Destination := value;
TryGetKeyUint := TRUE;
END_METHOD

METHOD TryGetKeyUlint : BOOL
VAR_INPUT
	Key : T_MAXSTRING;
	Destination : REFERENCE TO ULINT;
	Feedback : I_DeserializerFeedback;
END_VAR
VAR
	member : SJsonValue;
	value : ULINT;
	error : I_Error;
END_VAR
IF NOT TryGetMember(Key, member, Feedback) THEN
	RETURN;
END_IF

IF NOT TryReadNumber(member, value) THEN
	error := errorFactory.CreateIncorrectKeyTypeError('ULINT',Key);
	Feedback.LogError(error);
	RETURN;
END_IF

Destination := value;
TryGetKeyUlint := TRUE;
END_METHOD

METHOD TryGetKeyUsint : BOOL
VAR_INPUT
	Key : T_MAXSTRING;
	Destination : REFERENCE TO USINT;
	Feedback : I_DeserializerFeedback;
END_VAR
VAR
	member : SJsonValue;
	value : USINT;
	error : I_Error;
END_VAR
IF NOT TryGetMember(Key, member, Feedback) THEN
	RETURN;
END_IF

IF NOT TryReadNumber(member, value) THEN
	error := errorFactory.CreateIncorrectKeyTypeError('USINT',Key);
	Feedback.LogError(error);
	RETURN;
END_IF

Destination := value;
TryGetKeyUsint := TRUE;
END_METHOD

METHOD TryGetKeyWord : BOOL
VAR_INPUT
	Key : T_MAXSTRING;
	Destination : REFERENCE TO WORD;
	Feedback : I_DeserializerFeedback;
END_VAR
VAR
	member : SJsonValue;
	value : WORD;
	error : I_Error;
END_VAR
IF NOT TryGetMember(Key, member, Feedback) THEN
	RETURN;
END_IF

IF NOT TryReadNumber(member, value) THEN
	error := errorFactory.CreateIncorrectKeyTypeError('USINT',Key);
	Feedback.LogError(error);
	RETURN;
END_IF

Destination := value;
TryGetKeyWord := TRUE;
END_METHOD

METHOD TryGetLint : BOOL
VAR_INPUT
	Destination : REFERENCE TO LINT;
	Feedback : I_DeserializerFeedback;
END_VAR
VAR
	value : LINT;
	error : I_Error;
END_VAR
IF NOT TryReadNumber(root, value) THEN
	error := errorFactory.CreateIncorrectTypeError('LINT');
	Feedback.LogError(error);
	RETURN;
END_IF

Destination := value;
TryGetLint := TRUE;
END_METHOD

METHOD TryGetLreal : BOOL
VAR_INPUT
	Destination : REFERENCE TO LREAL;
	Feedback : I_DeserializerFeedback;
END_VAR
VAR
	value : LREAL;
	error : I_Error;
END_VAR
IF NOT TryReadNumber(root, value) THEN
	error := errorFactory.CreateIncorrectTypeError('LREAL');
	Feedback.LogError(error);
	RETURN;
END_IF

Destination := value;
TryGetLreal := TRUE;
END_METHOD

METHOD TryGetLtime : BOOL
VAR_INPUT
	Destination : REFERENCE TO LTIME;
	Feedback : I_DeserializerFeedback;
END_VAR
VAR
	timeAsString : T_MAXSTRING;
	error : I_Error;
END_VAR
IF NOT jsonParser.IsString(root) THEN
	error := errorFactory.CreateIncorrectTypeError('LTIME');
	Feedback.LogError(error);
	RETURN;
END_IF

timeAsString := jsonParser.GetString(root);
Destination := STRING_TO_LTIME(timeAsString);

TryGetLtime := TRUE;
END_METHOD

METHOD TryGetLword : BOOL
VAR_INPUT
	Destination : REFERENCE TO LWORD;
	Feedback : I_DeserializerFeedback;
END_VAR
VAR
	value : LWORD;
	error : I_Error;
END_VAR
IF NOT TryReadNumber(root, value) THEN
	error := errorFactory.CreateIncorrectTypeError('LWORD');
	Feedback.LogError(error);
	RETURN;
END_IF

Destination := value;
TryGetLword := TRUE;
END_METHOD

METHOD PROTECTED TryGetMember : BOOL
VAR_INPUT
	MemberName : T_MAXSTRING;
	Member : REFERENCE TO SJsonValue;
	Feedback : I_DeserializerFeedback;
END_VAR
VAR
	localMember : SJsonValue;
	error : I_Error;
END_VAR
IF MemberName = '' THEN
	error := errorFactory.CreateInvalidKeyError();
	Feedback.LogError(error);
	RETURN;
END_IF

localMember := jsonParser.FindMember(root, MemberName);

IF localMember = 0 THEN
	error := errorFactory.CreateMissingKeyError(MemberName);
	Feedback.LogError(error);
	RETURN;
END_IF

Member := localMember;
TryGetMember := TRUE;
END_METHOD

METHOD TryGetReal : BOOL
VAR_INPUT
	Destination : REFERENCE TO REAL;
	Feedback : I_DeserializerFeedback;
END_VAR
VAR
	value : REAL;
	error : I_Error;
END_VAR
IF NOT TryReadNumber(root, value) THEN
	error := errorFactory.CreateIncorrectTypeError('REAL');
	Feedback.LogError(error);
	RETURN;
END_IF

Destination := value;
TryGetReal := TRUE;
END_METHOD

METHOD TryGetSint : BOOL
VAR_INPUT
	Destination : REFERENCE TO SINT;
	Feedback : I_DeserializerFeedback;
END_VAR
VAR
	value : SINT;
	error : I_Error;
END_VAR
IF NOT TryReadNumber(root, value) THEN
	error := errorFactory.CreateIncorrectTypeError('SINT');
	Feedback.LogError(error);
	RETURN;
END_IF

Destination := value;
TryGetSint := TRUE;
END_METHOD

METHOD TryGetString : BOOL
VAR_INPUT
	Destination : REFERENCE TO T_MAXSTRING;
	Feedback : I_DeserializerFeedback;
END_VAR
VAR
	error : I_Error;
END_VAR
IF NOT TryReadString(root, Destination) THEN
	error := errorFactory.CreateIncorrectTypeError('STRING');
	Feedback.LogError(error);
	RETURN;
END_IF

TryGetString := TRUE;
END_METHOD

METHOD TryGetStringEx : BOOL
VAR_INPUT
	DestinationAddress : POINTER TO STRING;
	DestinationSize : UDINT;
	Feedback : I_DeserializerFeedback;
END_VAR
VAR
	error : I_Error;
END_VAR
IF NOT TryReadStringEx(root, DestinationAddress, DestinationSize) THEN
	error := errorFactory.CreateIncorrectTypeError('STRING');
	Feedback.LogError(error);
	RETURN;
END_IF

TryGetStringEx := TRUE;
END_METHOD

METHOD TryGetTime : BOOL
VAR_INPUT
	Destination : REFERENCE TO TIME;
	Feedback : I_DeserializerFeedback;
END_VAR
VAR
	timeAsString : T_MAXSTRING;
	error : I_Error;
END_VAR
IF NOT jsonParser.IsString(root) THEN
	error := errorFactory.CreateIncorrectTypeError('TIME');
	Feedback.LogError(error);
	RETURN;
END_IF

timeAsString := jsonParser.GetString(root);
Destination := STRING_TO_TIME(timeAsString);

TryGetTime := TRUE;
END_METHOD

METHOD TryGetTod : BOOL
VAR_INPUT
	Destination : REFERENCE TO TOD;
	Feedback : I_DeserializerFeedback;
END_VAR
VAR
	timeAsString : T_MAXSTRING;
	error : I_Error;
END_VAR
IF NOT jsonParser.IsString(root) THEN
	error := errorFactory.CreateIncorrectTypeError('TOD');
	Feedback.LogError(error);
	RETURN;
END_IF

timeAsString := jsonParser.GetString(root);
Destination := STRING_TO_TOD(timeAsString);

TryGetTod := TRUE;
END_METHOD

METHOD TryGetUdint : BOOL
VAR_INPUT
	Destination : REFERENCE TO UDINT;
	Feedback : I_DeserializerFeedback;
END_VAR
VAR
	value : UDINT;
	error : I_Error;
END_VAR
IF NOT TryReadNumber(root, value) THEN
	error := errorFactory.CreateIncorrectTypeError('UDINT');
	Feedback.LogError(error);
	RETURN;
END_IF

Destination := value;
TryGetUdint := TRUE;
END_METHOD

METHOD TryGetUint : BOOL
VAR_INPUT
	Destination : REFERENCE TO UINT;
	Feedback : I_DeserializerFeedback;
END_VAR
VAR
	value : UINT;
	error : I_Error;
END_VAR
IF NOT TryReadNumber(root, value) THEN
	error := errorFactory.CreateIncorrectTypeError('UINT');
	Feedback.LogError(error);
	RETURN;
END_IF

Destination := value;
TryGetUint := TRUE;
END_METHOD

METHOD TryGetUlint : BOOL
VAR_INPUT
	Destination : REFERENCE TO ULINT;
	Feedback : I_DeserializerFeedback;
END_VAR
VAR
	value : ULINT;
	error : I_Error;
END_VAR
IF NOT TryReadNumber(root, value) THEN
	error := errorFactory.CreateIncorrectTypeError('ULINT');
	Feedback.LogError(error);
	RETURN;
END_IF

Destination := value;
TryGetUlint := TRUE;
END_METHOD

METHOD TryGetUsint : BOOL
VAR_INPUT
	Destination : REFERENCE TO USINT;
	Feedback : I_DeserializerFeedback;
END_VAR
VAR
	value : USINT;
	error : I_Error;
END_VAR
IF NOT TryReadNumber(root, value) THEN
	error := errorFactory.CreateIncorrectTypeError('USINT');
	Feedback.LogError(error);
	RETURN;
END_IF

Destination := value;
TryGetUsint := TRUE;
END_METHOD

METHOD TryGetWord : BOOL
VAR_INPUT
	Destination : REFERENCE TO WORD;
	Feedback : I_DeserializerFeedback;
END_VAR
VAR
	value : WORD;
	error : I_Error;
END_VAR
IF NOT TryReadNumber(root, value) THEN
	error := errorFactory.CreateIncorrectTypeError('WORD');
	Feedback.LogError(error);
	RETURN;
END_IF

Destination := value;
TryGetWord := TRUE;
END_METHOD

METHOD PROTECTED TryReadBool : BOOL
VAR_INPUT
	JsonValue : SJsonValue;
	Destination : ANY;
END_VAR
VAR
	_BOOL : BOOL;
END_VAR
IF jsonValue = 0 THEN
	RETURN;
END_IF

IF jsonParser.IsBool(jsonValue) THEN
	_BOOL := jsonParser.GetBool(jsonValue);
	TryReadBool := TryConvert_BOOL_TO_DESTINATION(_BOOL,Destination);
	RETURN;
END_IF
END_METHOD

METHOD PROTECTED TryReadNumber : BOOL
VAR_INPUT
	JsonValue : SJsonValue;
	Destination : ANY;
END_VAR
VAR
	_DINT : DINT;
	_LINT : LINT;
	_UDINT : UDINT;
	_ULINT : ULINT;
	_LREAL : LREAL;
END_VAR
IF jsonValue = 0 THEN
	RETURN;
END_IF

IF jsonParser.IsInt(jsonValue) THEN
	_DINT := jsonParser.GetInt(jsonValue);
	TryReadNumber := TryConvert_DINT_TO_DESTINATION(_DINT,Destination);
	RETURN;
END_IF

IF jsonParser.IsInt64(jsonValue) THEN
	_LINT := jsonParser.GetInt64(jsonValue);
	TryReadNumber := TryConvert_LINT_TO_DESTINATION(_LINT,Destination);
	RETURN;
END_IF

IF jsonParser.IsUInt(jsonValue) THEN
	_UDINT := jsonParser.GetUInt(jsonValue);
	TryReadNumber := TryConvert_UDINT_TO_DESTINATION(_UDINT,Destination);
	RETURN;
END_IF

IF jsonParser.IsUInt64(jsonValue) THEN
	_ULINT := jsonParser.GetUInt64(jsonValue);
	TryReadNumber := TryConvert_ULINT_TO_DESTINATION(_ULINT,Destination);
	RETURN;
END_IF

IF jsonParser.IsDouble(jsonValue) THEN
	_LREAL := jsonParser.GetDouble(jsonValue);
	TryReadNumber := TryConvert_LREAL_TO_DESTINATION(_LREAL,Destination);
	RETURN;
END_IF
END_METHOD

METHOD PROTECTED TryReadString : BOOL
VAR_INPUT
	JsonValue : SJsonValue;
	Destination : REFERENCE TO T_MAXSTRING;
END_VAR
IF jsonValue = 0 THEN
	RETURN;
END_IF

IF jsonParser.IsString(jsonValue) THEN
	IF (jsonParser.CopyString(jsonValue,Destination,DINT_TO_UDINT(SIZEOF(Destination))) > 0) THEN;
		TryReadString := TRUE;
		RETURN;
	END_IF
END_IF
END_METHOD

METHOD PROTECTED TryReadStringEx : BOOL
VAR_INPUT
	JsonValue : SJsonValue;
	DestinationAddress : POINTER TO STRING;
	DestinationSize : UDINT;
END_VAR
IF jsonValue = 0 THEN
	RETURN;
END_IF

IF jsonParser.IsString(jsonValue) THEN
	IF (jsonParser.CopyString(jsonValue,DestinationAddress^,DestinationSize) > 0) THEN;
		TryReadStringEx := TRUE;
		RETURN;
	END_IF
END_IF
END_METHOD

END_FUNCTION_BLOCK

// ---- mobject-json/_Internal/JsonDeserializerForwardEnumerator/JsonDeserializerArrayForwardEnumerator.TcPOU
{attribute 'linkalways'} 
{attribute 'no_explicit_call' := 'This FB is a CLASS and must be accessed using methods or properties'}
{attribute 'enable_dynamic_creation'}
FUNCTION_BLOCK JsonDeserializerArrayForwardEnumerator EXTENDS Disposable IMPLEMENTS I_DeserializerArrayForwardEnumerator, I_EventHandler
VAR
	parent : I_JsonDeserializer;
	jsonParser : REFERENCE TO JsonDomParser;
	root : SJsonValue;
	garbageCollector : I_DeserializerGarbageCollector;
	nullNode : I_Deserializer;
	moveNextCalled : BOOL := FALSE;
	invalid : BOOL := FALSE; 
	nextArrayPosition : SJsonValue;
	arrayBeginPosition : SJsonValue;
	arrayEndPosition : SJsonValue;
	currentDeserializer : I_Deserializer;
	_index : DINT;
END_VAR

METHOD PROTECTED CreateDeserializer : I_Deserializer
VAR_INPUT
	DeserializerRoot : SJsonValue;
END_VAR
VAR 
	pNode : POINTER TO JsonDeserializerNode;
END_VAR
pNode := __NEW(JsonDeserializerNode(
	ParentJsonDeserializer := parent,
	ParentJsonDomParser := jsonParser, 
	NodeRoot := DeserializerRoot, 
	ParentGarbageCollector := garbageCollector, 
	ParentNullDeserializer := nullNode
));

CreateDeserializer := pNode^;
END_METHOD

PROPERTY PUBLIC Current : I_Deserializer
GET
IF NOT IsValid THEN
	Current := nullNode;
	RETURN;
END_IF

IF currentDeserializer = 0 THEN
	Current := nullNode;
	RETURN;
END_IF

Current := currentDeserializer;
END_GET
END_PROPERTY

METHOD FB_exit : BOOL
VAR_INPUT
	bInCopyCode : BOOL; // if TRUE, the exit method is called for exiting an instance that is copied afterwards (online change).
END_VAR
IF bInCopyCode THEN
	RETURN;
END_IF

IF parent = 0 THEN
	RETURN;
END_IF

parent.OffEvent('OnChanged',THIS^);
parent.OffEvent('OnDisposed',THIS^);
END_METHOD

METHOD FB_init : BOOL
VAR_INPUT
	bInitRetains : BOOL; // if TRUE, the retain variables are initialized (warm start / cold start)
	bInCopyCode : BOOL;  // if TRUE, the instance afterwards gets moved into the copy code (online change)
	ParentJsonDeserializer : I_JsonDeserializer;
	ParentJsonDomParser : REFERENCE TO JsonDomParser;
	NodeRoot : SJsonValue;
	ParentGarbageCollector : I_DeserializerGarbageCollector;
	ParentNullDeserializer : I_Deserializer;
END_VAR
THIS^.parent := ParentJsonDeserializer;
THIS^.jsonParser REF= ParentJsonDomParser;
THIS^.root := NodeRoot;
THIS^.garbageCollector := ParentGarbageCollector;
THIS^.nullNode := ParentNullDeserializer;

Initialize();

Parent.OnEvent('OnChanged',THIS^);
Parent.OnEvent('OnDisposed',THIS^);
END_METHOD

METHOD PUBLIC HandleEvent
VAR_INPUT
	Event : I_Event;
END_VAR
VAR
	changedEvent : I_JsonDeserializerChangedEvent;
	disposedEvent : I_JsonDeserializerDisposedEvent;
END_VAR
IF __QUERYINTERFACE(Event, changedEvent) THEN
	invalid := TRUE;
ELSIF __QUERYINTERFACE(Event, disposedEvent) THEN
	parent := 0;
	Dispose();
END_IF
END_METHOD

PROPERTY Index : DINT
GET
Index := _index;
END_GET
END_PROPERTY

METHOD PROTECTED Initialize
VAR_INPUT
END_VAR
IF NOT jsonParser.IsArray(root) THEN
	invalid := TRUE;
	RETURN;
END_IF

arrayBeginPosition := jsonParser.ArrayBegin(root);
arrayEndPosition := jsonParser.ArrayEnd(root);

IF arrayBeginPosition = 0 THEN
	invalid := TRUE;
	RETURN;
END_IF

IF arrayEndPosition = 0 THEN
	invalid := TRUE;
	RETURN;
END_IF
END_METHOD

PROPERTY PUBLIC IsValid : BOOL
GET // PUBLIC
IF invalid THEN
	RETURN;
END_IF

IF parent = 0 THEN
	RETURN;
END_IF

IsValid := TRUE;
END_GET
END_PROPERTY

METHOD PUBLIC MoveNext : BOOL
IF invalid THEN
    RETURN;
END_IF

// Handle the initial move
IF NOT moveNextCalled THEN
    moveNextCalled := TRUE;
    UpdateCurrentDeserializer(arrayBeginPosition);
	nextArrayPosition := jsonParser.NextArray(arrayBeginPosition);
	_index := _index + 1;
	MoveNext := TRUE;
    RETURN;
END_IF

// Handle subsequent moves
IF nextArrayPosition <> arrayEndPosition THEN
	UpdateCurrentDeserializer(nextArrayPosition);
	nextArrayPosition := jsonParser.NextArray(nextArrayPosition);
	_index := _index + 1;
	MoveNext := TRUE;
END_IF
END_METHOD

METHOD PROTECTED UpdateCurrentDeserializer
VAR_INPUT
	Root : SJsonValue;
END_VAR
VAR
	newRoot : SJsonValue;
END_VAR
IF currentDeserializer <> 0 THEN
	currentDeserializer.Dispose();
	currentDeserializer := 0;
END_IF

IF invalid THEN
	RETURN;
END_IF

newRoot := jsonParser.GetArrayValue(Root);

IF newRoot = 0 THEN
	RETURN;
END_IF

currentDeserializer := CreateDeserializer(newRoot);
END_METHOD

END_FUNCTION_BLOCK

// ---- mobject-json/_Internal/JsonDeserializerForwardEnumerator/JsonDeserializerObjectForwardEnumerator.TcPOU
{attribute 'linkalways'} 
{attribute 'no_explicit_call' := 'This FB is a CLASS and must be accessed using methods or properties'}
{attribute 'enable_dynamic_creation'}
FUNCTION_BLOCK JsonDeserializerObjectForwardEnumerator EXTENDS Disposable IMPLEMENTS I_DeserializerObjectForwardEnumerator, I_EventHandler
VAR
	parent : I_JsonDeserializer;
	jsonParser : REFERENCE TO JsonDomParser;
	root : SJsonValue;
	garbageCollector : I_DeserializerGarbageCollector;
	nullNode : I_Deserializer;
	moveNextCalled : BOOL := FALSE;
	invalid : BOOL := FALSE; 
	nextMemberPosition : SJsonValue;
	memberBeginPosition : SJsonValue;
	memberEndPosition : SJsonValue;
	currentDeserializer : I_Deserializer;
	currentKey : T_MAXSTRING;
END_VAR

METHOD PROTECTED CreateDeserializer : I_Deserializer
VAR_INPUT
	DeserializerRoot : SJsonValue;
END_VAR
VAR 
	pNode : POINTER TO JsonDeserializerNode;
END_VAR
pNode := __NEW(JsonDeserializerNode(
	ParentJsonDeserializer := parent,
	ParentJsonDomParser := jsonParser, 
	NodeRoot := DeserializerRoot, 
	ParentGarbageCollector := garbageCollector, 
	ParentNullDeserializer := nullNode
));

CreateDeserializer := pNode^;
END_METHOD

PROPERTY PUBLIC Current : I_Deserializer
GET
IF NOT IsValid THEN
	Current := nullNode;
	RETURN;
END_IF

IF currentDeserializer = 0 THEN
	Current := nullNode;
	RETURN;
END_IF

Current := currentDeserializer;
END_GET
END_PROPERTY

METHOD FB_exit : BOOL
VAR_INPUT
	bInCopyCode : BOOL; // if TRUE, the exit method is called for exiting an instance that is copied afterwards (online change).
END_VAR
IF bInCopyCode THEN
	RETURN;
END_IF

IF parent = 0 THEN
	RETURN;
END_IF

parent.OffEvent('OnChanged',THIS^);
parent.OffEvent('OnDisposed',THIS^);
END_METHOD

METHOD FB_init : BOOL
VAR_INPUT
	bInitRetains : BOOL; // if TRUE, the retain variables are initialized (warm start / cold start)
	bInCopyCode : BOOL;  // if TRUE, the instance afterwards gets moved into the copy code (online change)
	ParentJsonDeserializer : I_JsonDeserializer;
	ParentJsonDomParser : REFERENCE TO JsonDomParser;
	NodeRoot : SJsonValue;
	ParentGarbageCollector : I_DeserializerGarbageCollector;
	ParentNullDeserializer : I_Deserializer;
END_VAR
THIS^.parent := ParentJsonDeserializer;
THIS^.jsonParser REF= ParentJsonDomParser;
THIS^.root := NodeRoot;
THIS^.garbageCollector := ParentGarbageCollector;
THIS^.nullNode := ParentNullDeserializer;

Initialize();

Parent.OnEvent('OnChanged',THIS^);
Parent.OnEvent('OnDisposed',THIS^);
END_METHOD

METHOD PUBLIC HandleEvent
VAR_INPUT
	Event : I_Event;
END_VAR
VAR
	changedEvent : I_JsonDeserializerChangedEvent;
	disposedEvent : I_JsonDeserializerDisposedEvent;
END_VAR
IF __QUERYINTERFACE(Event, changedEvent) THEN
	invalid := TRUE;
ELSIF __QUERYINTERFACE(Event, disposedEvent) THEN
	parent := 0;
	Dispose();
END_IF
END_METHOD

METHOD PROTECTED Initialize
VAR_INPUT
END_VAR
IF NOT jsonParser.IsObject(root) THEN
	invalid := TRUE;
	RETURN;
END_IF

memberBeginPosition := jsonParser.MemberBegin(root);
memberEndPosition := jsonParser.MemberEnd(root);

IF memberBeginPosition = 0 THEN
	invalid := TRUE;
	RETURN;
END_IF

IF memberEndPosition = 0 THEN
	invalid := TRUE;
	RETURN;
END_IF
END_METHOD

PROPERTY PUBLIC IsValid : BOOL
GET // PUBLIC
IF invalid THEN
	RETURN;
END_IF

IF parent = 0 THEN
	RETURN;
END_IF

IsValid := TRUE;
END_GET
END_PROPERTY

PROPERTY Key : T_MAXSTRING
GET
Key := currentKey;
END_GET
END_PROPERTY

METHOD PUBLIC MoveNext : BOOL
IF invalid THEN
    RETURN;
END_IF

// Handle the initial move
IF NOT moveNextCalled THEN
    moveNextCalled := TRUE;
    UpdateCurrentDeserializer(memberBeginPosition);
	nextMemberPosition := jsonParser.NextMember(memberBeginPosition);
	MoveNext := TRUE;
    RETURN;
END_IF

// Handle subsequent moves
IF nextMemberPosition <> memberEndPosition THEN	
	UpdateCurrentDeserializer(nextMemberPosition);
	nextMemberPosition := jsonParser.NextMember(nextMemberPosition);
	MoveNext := TRUE;
END_IF
END_METHOD

METHOD PROTECTED UpdateCurrentDeserializer
VAR_INPUT
	UpdatedRoot : SJsonValue;
END_VAR
VAR
	rootOfValue : SJsonValue;
END_VAR
IF currentDeserializer <> 0 THEN
	currentDeserializer.Dispose();
	currentDeserializer := 0;
END_IF

IF invalid THEN
	RETURN;
END_IF

rootOfValue := jsonParser.GetMemberValue(UpdatedRoot);
currentKey := jsonParser.GetMemberName(UpdatedRoot);

IF rootOfValue = 0 THEN
	RETURN;
END_IF

currentDeserializer := CreateDeserializer(rootOfValue);
END_METHOD

END_FUNCTION_BLOCK

// ---- mobject-json/_Internal/Events/JsonDeserializerChangedEvent.TcPOU
{attribute 'linkalways'} 
{attribute 'no_explicit_call' := 'This FB is a CLASS and must be accessed using methods or properties'}
{attribute 'enable_dynamic_creation'}
FUNCTION_BLOCK JsonDeserializerChangedEvent EXTENDS JsonDeserializerEvent IMPLEMENTS I_JsonDeserializerChangedEvent

END_FUNCTION_BLOCK

// ---- mobject-json/_Internal/Events/JsonDeserializerEvent.TcPOU
{attribute 'linkalways'} 
{attribute 'no_explicit_call' := 'This FB is a CLASS and must be accessed using methods or properties'}
{attribute 'enable_dynamic_creation'}
FUNCTION_BLOCK ABSTRACT JsonDeserializerEvent EXTENDS Disposable
VAR
	_target : I_JsonDeserializer;
END_VAR

METHOD FB_init : BOOL
VAR_INPUT
	bInitRetains : BOOL; // if TRUE, the retain variables are initialized (warm start / cold start)
	bInCopyCode : BOOL;  // if TRUE, the instance afterwards gets moved into the copy code (online change)
	Target : I_JsonDeserializer;
END_VAR
This^._target := Target;
END_METHOD

PROPERTY PUBLIC Target : I_JsonDeserializer
GET // PUBLIC
Target := _target;
END_GET
END_PROPERTY

END_FUNCTION_BLOCK

// ---- mobject-json/JsonSerializer/JsonSerializer.TcPOU
{attribute 'linkalways'} 
{attribute 'no_explicit_call' := 'This FB is a CLASS and must be accessed using methods or properties'}
{attribute 'enable_dynamic_creation'}
FUNCTION_BLOCK JsonSerializer EXTENDS Disposable IMPLEMENTS I_Serializer;
VAR
	jsonSaxWriter : FB_JsonSaxWriter;
END_VAR

METHOD PUBLIC AddBase64 : I_Serializer
VAR_INPUT
	pBytes : POINTER TO BYTE;
	nBytes : DINT;
END_VAR
jsonSaxWriter.AddBase64(pBytes, nBytes);
AddBase64 := THIS^;
END_METHOD

METHOD PUBLIC AddBool : I_Serializer
VAR_INPUT
	Value : BOOL;
END_VAR
jsonSaxWriter.AddBool(Value);
AddBool := THIS^;
END_METHOD

METHOD PUBLIC AddByte : I_Serializer
VAR_INPUT
	Value : BYTE;
END_VAR
jsonSaxWriter.AddUDint(BYTE_TO_UDINT(Value));
AddByte := THIS^;
END_METHOD

METHOD PUBLIC AddBytesAsHex : I_Serializer
VAR_INPUT
	pBytes : POINTER TO BYTE;
	nBytes : DINT;
END_VAR
jsonSaxWriter.AddHexBinary(pBytes, nBytes);
AddBytesAsHex := THIS^;
END_METHOD

METHOD PUBLIC AddDateTime : I_Serializer
VAR_INPUT
	Value : DATE_AND_TIME;
END_VAR
jsonSaxWriter.AddDateTime(Value);
AddDateTime := THIS^;
END_METHOD

METHOD PUBLIC AddDcTime : I_Serializer
VAR_INPUT
	Value : DCTIME;
END_VAR
jsonSaxWriter.AddDcTime(Value);
AddDcTime := THIS^;
END_METHOD

METHOD PUBLIC AddDint : I_Serializer
VAR_INPUT
	Value : DINT;
END_VAR
jsonSaxWriter.AddDint(Value);
AddDint := THIS^;
END_METHOD

METHOD PUBLIC AddDword : I_Serializer
VAR_INPUT
	Value : DWORD;
END_VAR
jsonSaxWriter.AddUDint(DWORD_TO_UDINT(Value));
AddDword := THIS^;
END_METHOD

METHOD PUBLIC AddFileTime : I_Serializer
VAR_INPUT
	Value : FILETIME;
END_VAR
jsonSaxWriter.AddFileTime(Value);
AddFileTime := THIS^;
END_METHOD

METHOD PUBLIC AddInt : I_Serializer
VAR_INPUT
	Value : INT;
END_VAR
jsonSaxWriter.AddDint(INT_TO_DINT(Value));
AddInt := THIS^;
END_METHOD

METHOD PUBLIC AddKey : I_Serializer
VAR_INPUT
	Key : T_MAXSTRING;
END_VAR
jsonSaxWriter.AddKey(Key);
AddKey := THIS^;
END_METHOD

METHOD PUBLIC AddKeyBase64 : I_Serializer
VAR_INPUT
	Key : T_MAXSTRING;
	pBytes : POINTER TO BYTE;
	nBytes : DINT;
END_VAR
AddKey(Key);
AddBase64(pBytes, nBytes);
AddKeyBase64 := THIS^;
END_METHOD

METHOD PUBLIC AddKeyBool : I_Serializer
VAR_INPUT
	Key : T_MAXSTRING;
	Value : BOOL;
END_VAR
AddKey(Key);
AddBool(Value);
AddKeyBool := THIS^;
END_METHOD

METHOD PUBLIC AddKeyByte : I_Serializer
VAR_INPUT
	Key : T_MAXSTRING;
	Value : BYTE;
END_VAR
AddKey(Key);
AddByte(Value);
AddKeyByte := THIS^;
END_METHOD

METHOD PUBLIC AddKeyBytesAsHex : I_Serializer
VAR_INPUT
	Key : T_MAXSTRING;
	pBytes : POINTER TO BYTE;
	nBytes : DINT;
END_VAR
AddKey(Key);
AddBytesAsHex(pBytes, nBytes);
AddKeyBytesAsHex := THIS^;
END_METHOD

METHOD PUBLIC AddKeyDateTime : I_Serializer
VAR_INPUT
	Key : T_MAXSTRING;
	Value : DATE_AND_TIME;
END_VAR
AddKey(Key);
AddDateTime(Value);
AddKeyDateTime := THIS^;
END_METHOD

METHOD PUBLIC AddKeyDcTime : I_Serializer
VAR_INPUT
	Key : T_MAXSTRING;
	Value : DCTIME;
END_VAR
AddKey(Key);
AddDcTime(Value);
AddKeyDcTime := THIS^;
END_METHOD

METHOD PUBLIC AddKeyDint : I_Serializer
VAR_INPUT
	Key : T_MAXSTRING;
	Value : DINT;
END_VAR
AddKey(Key);
AddDint(Value);
AddKeyDint := THIS^;
END_METHOD

METHOD PUBLIC AddKeyDword : I_Serializer
VAR_INPUT
	Key : T_MAXSTRING;
	Value : DWORD;
END_VAR
AddKey(Key);
AddDword(Value);
AddKeyDword := THIS^;
END_METHOD

METHOD PUBLIC AddKeyFileTime : I_Serializer
VAR_INPUT
	Key : T_MAXSTRING;
	Value : FILETIME;
END_VAR
AddKey(Key);
AddFileTime(Value);
AddKeyFileTime := THIS^;
END_METHOD

METHOD PUBLIC AddKeyInt : I_Serializer
VAR_INPUT
	Key : T_MAXSTRING;
	Value : INT;
END_VAR
AddKey(Key);
AddInt(Value);
AddKeyInt := THIS^;
END_METHOD

METHOD PUBLIC AddKeyLint : I_Serializer
VAR_INPUT
	Key : T_MAXSTRING;
	Value : LINT;
END_VAR
AddKey(Key);
AddLint(Value);
AddKeyLint := THIS^;
END_METHOD

METHOD PUBLIC AddKeyLreal : I_Serializer
VAR_INPUT
	Key : T_MAXSTRING;
	Value : LREAL;
END_VAR
AddKey(Key);
AddLreal(Value);
AddKeyLreal := THIS^;
END_METHOD

METHOD PUBLIC AddKeyLtime : I_Serializer
VAR_INPUT
	Key : T_MAXSTRING;
	Value : LTIME;
END_VAR
AddKey(Key);
AddLTIME(Value);
AddKeyLtime := THIS^;
END_METHOD

METHOD PUBLIC AddKeyLword : I_Serializer
VAR_INPUT
	Key : T_MAXSTRING;
	Value : LWORD;
END_VAR
AddKey(Key);
AddLword(Value);
AddKeyLword := THIS^;
END_METHOD

METHOD PUBLIC AddKeyNull : I_Serializer
VAR_INPUT
	Key : T_MAXSTRING;
END_VAR
AddKey(Key);
AddNull();
AddKeyNull := THIS^;
END_METHOD

METHOD PUBLIC AddKeyObject : I_Serializer
VAR_INPUT
	Key : T_MAXSTRING;
	Object : I_Serializable;
END_VAR
AddKey(Key);
Object.SerializeWith(THIS^);
AddKeyObject := THIS^;
END_METHOD

METHOD PUBLIC AddKeyRawJson : I_Serializer
VAR_INPUT
	Key : T_MAXSTRING;
	RawObject : REFERENCE TO STRING;;
END_VAR
AddKey(Key);
AddRawJson(RawObject);
AddKeyRawJson := THIS^;
END_METHOD

METHOD PUBLIC AddKeyReal : I_Serializer
VAR_INPUT
	Key : T_MAXSTRING;
	Value : REAL;
END_VAR
AddKey(Key);
AddReal(Value);
AddKeyReal := THIS^;
END_METHOD

METHOD PUBLIC AddKeySint : I_Serializer
VAR_INPUT
	Key : T_MAXSTRING;
	Value : SINT;
END_VAR
AddKey(Key);
AddSint(Value);
AddKeySint := THIS^;
END_METHOD

METHOD PUBLIC AddKeyString : I_Serializer
VAR_INPUT
	Key : T_MAXSTRING;
	Value : T_MAXSTRING;
END_VAR
AddKey(Key);
AddString(Value);
AddKeyString := THIS^;
END_METHOD

METHOD PUBLIC AddKeyStringByRef : I_Serializer
VAR_INPUT
	Key : T_MAXSTRING;
	Value : REFERENCE TO STRING;;
END_VAR
AddKey(Key);
AddStringByRef(Value);
AddKeyStringByRef := THIS^;
END_METHOD

METHOD PUBLIC AddKeyTime : I_Serializer
VAR_INPUT
	Key : T_MAXSTRING;
	Value : TIME;
END_VAR
AddKey(Key);
AddTime(Value);
AddKeyTime := THIS^;
END_METHOD

METHOD PUBLIC AddKeyTod : I_Serializer
VAR_INPUT
	Key : T_MAXSTRING;
	Value : TOD;
END_VAR
AddKey(Key);
AddTod(Value);
AddKeyTod := THIS^;
END_METHOD

METHOD PUBLIC AddKeyUdint : I_Serializer
VAR_INPUT
	Key : T_MAXSTRING;
	Value : UDINT;
END_VAR
AddKey(Key);
AddUdint(Value);
AddKeyUdint := THIS^;
END_METHOD

METHOD PUBLIC AddKeyUint : I_Serializer
VAR_INPUT
	Key : T_MAXSTRING;
	Value : UINT;
END_VAR
AddKey(Key);
AddUint(Value);
AddKeyUint := THIS^;
END_METHOD

METHOD PUBLIC AddKeyUlint : I_Serializer
VAR_INPUT
	Key : T_MAXSTRING;
	Value : ULINT;
END_VAR
AddKey(Key);
AddUlint(Value);
AddKeyUlint := THIS^;
END_METHOD

METHOD PUBLIC AddKeyUsint : I_Serializer
VAR_INPUT
	Key : T_MAXSTRING;
	Value : USINT;
END_VAR
AddKey(Key);
AddUsint(Value);
AddKeyUsint := THIS^;
END_METHOD

METHOD PUBLIC AddKeyWord : I_Serializer
VAR_INPUT
	Key : T_MAXSTRING;
	Value : WORD;
END_VAR
AddKey(Key);
AddWord(Value);
AddKeyWord := THIS^;
END_METHOD

METHOD PUBLIC AddLint : I_Serializer
VAR_INPUT
	Value : LINT;
END_VAR
jsonSaxWriter.AddLint(Value);
AddLint := THIS^;
END_METHOD

METHOD PUBLIC AddLreal : I_Serializer
VAR_INPUT
	Value : LREAL;
END_VAR
jsonSaxWriter.AddLreal(Value);
AddLreal := THIS^;
END_METHOD

METHOD PUBLIC AddLtime : I_Serializer
VAR_INPUT
	Value : LTIME;
END_VAR
VAR
	converted : T_MAXSTRING;
END_VAR
converted := LTIME_TO_STRING(Value);
jsonSaxWriter.AddString(converted);
AddLtime := THIS^;
END_METHOD

METHOD PUBLIC AddLword : I_Serializer
VAR_INPUT
	Value : LWORD;
END_VAR
jsonSaxWriter.AddUlint(LWORD_TO_ULINT(Value));
AddLword := THIS^;
END_METHOD

METHOD PUBLIC AddNull : I_Serializer
VAR_INPUT
END_VAR
jsonSaxWriter.AddNull();
AddNull := THIS^;
END_METHOD

METHOD PUBLIC AddObject
VAR_INPUT
	Object : I_Serializable;
END_VAR
Object.SerializeWith(This^);
END_METHOD

METHOD PUBLIC AddRawJson
VAR_INPUT
	RawObject : REFERENCE TO STRING;
END_VAR
jsonSaxWriter.AddRawObject(RawObject);
END_METHOD

METHOD PUBLIC AddReal : I_Serializer
VAR_INPUT
	Value : REAL;
END_VAR
// real to lreal is used to negate an issue with TC4024.55 which prevents max REAL from being serailized.  
// so a REAL_TO_LREAL conversion is made to ensure this is always possible.  
jsonSaxWriter.AddLReal(REAL_TO_LREAL(Value));
AddReal := THIS^;
END_METHOD

METHOD PUBLIC AddSint : I_Serializer
VAR_INPUT
	Value : SINT;
END_VAR
jsonSaxWriter.AddDint(SINT_TO_DINT(Value));
AddSint := THIS^;
END_METHOD

METHOD PUBLIC AddString : I_Serializer
VAR_INPUT
	Value : T_MAXSTRING;
END_VAR
jsonSaxWriter.AddString(Value);
AddString := THIS^;
END_METHOD

METHOD PUBLIC AddStringByRef : I_Serializer
VAR_INPUT
	Value : REFERENCE TO STRING;
END_VAR
jsonSaxWriter.AddString(Value);
AddStringByRef := THIS^;
END_METHOD

METHOD PUBLIC AddTime : I_Serializer
VAR_INPUT
	Value : TIME;
END_VAR
VAR
	converted : T_MAXSTRING;
END_VAR
converted := TIME_TO_STRING(Value);
jsonSaxWriter.AddString(converted);
AddTime := THIS^;
END_METHOD

METHOD PUBLIC AddTod : I_Serializer
VAR_INPUT
	Value : TOD;
END_VAR
VAR
	converted : T_MAXSTRING;
END_VAR
converted := TOD_TO_STRING(Value);
jsonSaxWriter.AddString(converted);
AddTod := THIS^;
END_METHOD

METHOD PUBLIC AddUdint : I_Serializer
VAR_INPUT
	Value : UDINT;
END_VAR
jsonSaxWriter.AddUdint(Value);
AddUdint := THIS^;
END_METHOD

METHOD PUBLIC AddUint : I_Serializer
VAR_INPUT
	Value : UINT;
END_VAR
jsonSaxWriter.AddDint(UINT_TO_DINT(Value));
AddUint := THIS^;
END_METHOD

METHOD PUBLIC AddUlint : I_Serializer
VAR_INPUT
	Value : ULINT;
END_VAR
jsonSaxWriter.AddUlint(Value);
AddUlint := THIS^;
END_METHOD

METHOD PUBLIC AddUsint : I_Serializer
VAR_INPUT
	Value : USINT;
END_VAR
jsonSaxWriter.AddDint(USINT_TO_DINT(Value));
AddUsint := THIS^;
END_METHOD

METHOD PUBLIC AddWord : I_Serializer
VAR_INPUT
	Value : WORD;
END_VAR
jsonSaxWriter.AddUDint(WORD_TO_UDINT(Value));
AddWord := THIS^;
END_METHOD

METHOD PUBLIC Clone : I_Serializer
VAR
	pClone : POINTER TO JsonSerializer;
	jsonSize : UDINT;
	pJsonString : POINTER TO STRING;
END_VAR
pClone := __NEW(JsonSerializer);
Clone := pClone^;

jsonSize := jsonSaxWriter.GetDocumentLength();

IF jsonSize = 0 THEN
	// no further cloning to do. 
	RETURN;
END_IF

pJsonString := __NEW(BYTE, jsonSize);

IF jsonSaxWriter.CopyDocument(pJsonString^, jsonSize) = 0 THEN
	__DELETE(pJsonString);
	RETURN;
END_IF

pClone^.AddRawJson(pJsonString^);
__DELETE(pJsonString);
END_METHOD

METHOD PUBLIC EndArray : I_Serializer
VAR_INPUT
END_VAR
jsonSaxWriter.EndArray();
EndArray := THIS^;
END_METHOD

METHOD PUBLIC EndObject : I_Serializer
VAR_INPUT
END_VAR
jsonSaxWriter.EndObject();
EndObject := THIS^;
END_METHOD

METHOD FB_exit : BOOL
VAR_INPUT
	bInCopyCode : BOOL; // if TRUE, the exit method is called for exiting an instance that is copied afterwards (online change).
END_VAR
IF bInCopyCode THEN
	RETURN;
END_IF

jsonSaxWriter.ResetDocument();
END_METHOD

METHOD PUBLIC GetSerializedDataLength : UDINT
VAR_INPUT
END_VAR
GetSerializedDataLength := jsonSaxWriter.GetDocumentLength();
END_METHOD

METHOD PUBLIC Reset
VAR_INPUT
END_VAR
jsonSaxWriter.ResetDocument();
END_METHOD

METHOD PUBLIC StartArray : I_Serializer
VAR_INPUT
END_VAR
jsonSaxWriter.StartArray();
StartArray := THIS^;
END_METHOD

METHOD PUBLIC StartObject : I_Serializer
VAR_INPUT
END_VAR
jsonSaxWriter.StartObject();
StartObject := THIS^;
END_METHOD

METHOD TryCopySerializedData : BOOL
VAR_INPUT
	DestinationAddress : PVOID;
	DestinationSize : UDINT;
END_VAR
VAR
	pString : POINTER TO STRING;
END_VAR
pString := DestinationAddress;
TryCopySerializedData := jsonSaxWriter.CopyDocument(pString^, DestinationSize) > 0;
END_METHOD

METHOD TryGetSerializedData : BOOL
VAR_INPUT
	DestinationAddress : PVOID;
	DestinationSize : UDINT;
END_VAR
VAR
	pString : POINTER TO STRING;
END_VAR
pString := DestinationAddress;

IF jsonSaxWriter.CopyDocument(pString^, DestinationSize) = 0 THEN
	RETURN;
END_IF

jsonSaxWriter.ResetDocument();
TryGetSerializedData := TRUE;
END_METHOD

END_FUNCTION_BLOCK

// ---- mobject-server/RpcHandler/Examples/AsyncConcatStringRpcHandler.TcPOU
{attribute 'linkalways'} 
FUNCTION_BLOCK AsyncConcatStringRpcHandler IMPLEMENTS I_AsynchronousRpcHandler
VAR
END_VAR

METHOD Handle
VAR_INPUT
	Parameters : I_Deserializer;
	Response : I_AsynchronousRpcResponse;
END_VAR
VAR
	str1 : T_MAXSTRING;
	str2 : T_MAXSTRING;
	result : T_MAXSTRING;
	feedback : DeserializerFeedback;
END_VAR
IF NOT Parameters.TryGetKeyString('STR1',str1,feedback) THEN
	Response.RejectWithError('MISSING_PARAMETER',feedback.FirstError.Message);
	RETURN;
END_IF

IF NOT Parameters.TryGetKeyString('STR2',str2,feedback) THEN
	Response.RejectWithError('MISSING_PARAMETER',feedback.FirstError.Message);
	RETURN;
END_IF

result := CONCAT(str1, str2);
Response.CompleteWithString(result);
END_METHOD

END_FUNCTION_BLOCK

// ---- mobject-server/RpcHandler/Examples/ConcatStringRpcHandler.TcPOU
{attribute 'linkalways'} 
FUNCTION_BLOCK ConcatStringRpcHandler IMPLEMENTS I_SynchronousRpcHandler
VAR
END_VAR

METHOD Handle
VAR_INPUT
	Parameters : I_Deserializer;
	Response : I_SynchronousRpcResponse;
END_VAR
VAR
	str1 : T_MAXSTRING;
	str2 : T_MAXSTRING;
	result : T_MAXSTRING;
	feedback : DeserializerFeedback;
END_VAR
IF NOT Parameters.TryGetKeyString('STR1',str1,feedback) THEN
	Response.RejectWithError('MISSING_PARAMETER',feedback.FirstError.Message);
	RETURN;
END_IF

IF NOT Parameters.TryGetKeyString('STR2',str2,feedback) THEN
	Response.RejectWithError('MISSING_PARAMETER',feedback.FirstError.Message);
	RETURN;
END_IF

result := CONCAT(str1, str2);
Response.CompleteWithString(result);
END_METHOD

END_FUNCTION_BLOCK

// ---- mobject-server/RpcServer/RpcServer.TcPOU
{attribute 'linkalways'} 
{attribute 'no_explicit_call' := 'This FB is a CLASS and must be accessed using methods or properties'}
{attribute 'enable_dynamic_creation'}
{attribute 'TcRpcEnable'}
FUNCTION_BLOCK RpcServer IMPLEMENTS I_RpcServer
VAR
	// default header accessor.
	headerAccessor : HeaderAccessor;
	
	// Payload size may be changed using the constants
	payloadStringSizeIncludingNull : UDINT := ServerConfiguration.PAYLOAD_STRING_SIZE + 1;
	
	// the middleware stack allows us to construct our server in any way needed.
	// by default we will support sessions, async polling and chunked requests/
	middlewareStack : MiddlewareStack;
	
	// responseId generation required for pending or chunked data
	sequentialResponseIdGenerator : SequentialResponseIdGenerator;
	
	// ability to support sessions...
	sessionIdGenerator : SequentialSessionIdGenerator;
	sessionManager : SessionManager(sessionIdGenerator, INACTIVE_SESSION_MAX_AGE);
	sessionsMiddleware : SessionsMiddleware(sessionManager, headerAccessor);
	
	// ability to suppoort chunked requests
	chunkedRequestsManager : ChunkedRequestsManager(payloadStringSizeIncludingNull, sessionManager, headerAccessor);
	chunkedRequestsMiddleware : ChunkedRequestsMiddleware(chunkedRequestsManager);
	
	// ability to support chunked responses
	chunkedResponseManager : ChunkedResponseManager(payloadStringSizeIncludingNull, sessionManager, sequentialResponseIdGenerator, headerAccessor);
	chunkedResponsesMiddleware : ChunkedResponsesMiddleware(chunkedResponseManager);
	
	// ability to support pending responses
	asyncResponseManager : AsyncResponseManager(sessionManager, sequentialResponseIdGenerator, headerAccessor, ServerConfiguration.PENDING_RESPONSE_MAX_AGE);
	asyncResponseMiddleware : AsyncResponseMiddleware(asyncResponseManager);
	
	// guard
	responseIdGuardMiddleware : ResponseIdGuardMiddleware(headerAccessor);
	
	// ability to support rpc
	synchronousRpcHandlers : SynchronousRpcHandlers;
	asynchronousRpcHandlers : AsynchronousRpcHandlers;
	asyncRpcCallQueue : AsyncRpcCallQueue;
	rpcManager : RpcManager(synchronousRpcHandlers, asynchronousRpcHandlers, asyncResponseManager, headerAccessor, asyncRpcCallQueue);
	rpcMiddleware : RpcMiddleware(rpcManager);
	
	// registered apis (used for cyclic calling)
	registeredRpcApis : RegisteredRpcApis;
	
END_VAR
VAR CONSTANT
	INACTIVE_SESSION_MAX_AGE : TIME := T#10S;
END_VAR

METHOD PUBLIC CyclicCall
VAR_INPUT
END_VAR
sessionManager.CyclicCall();
asyncRpcCallQueue.CyclicCall();
registeredRpcApis.CyclicCall();
END_METHOD

METHOD FB_init : BOOL
VAR_INPUT
	bInitRetains : BOOL; // if TRUE, the retain variables are initialized (warm start / cold start)
	bInCopyCode : BOOL;  // if TRUE, the instance afterwards gets moved into the copy code (online change)
END_VAR
// must be above any middleware which requires storing of session data. 
// best practice is to put at the top
MiddlewareStack.Use(sessionsMiddleware);

// must be above any middleware which could send a response larger than the max payload.
// once this is in place then middleware can send as large as they like (up to router memory max)
MiddlewareStack.Use(chunkedResponsesMiddleware);

// must be above any middleware which needs to support async responses
MiddlewareStack.Use(AsyncResponseMiddleware);

// Any Response-Id reaching here was not recognised by either
// response middleware and must not be allowed to reach RPC.
MiddlewareStack.Use(responseIdGuardMiddleware);

// chunked request must be after chunked response to prevent incorrectly starting a new request
// if the client askes for a response without removing the last request header.
MiddlewareStack.Use(chunkedRequestsMiddleware); 

// rpc middlware.  All other middleware can go under here.
MiddlewareStack.Use(rpcMiddleware);
END_METHOD

{attribute 'TcRpcEnable'}
METHOD PUBLIC GetConfiguredHeaderSize : UDINT
VAR_INPUT
END_VAR
GetConfiguredHeaderSize := ServerConfiguration.HEADER_STRING_SIZE;
END_METHOD

{attribute 'TcRpcEnable'}
METHOD PUBLIC GetConfiguredPayloadSize : UDINT
VAR_INPUT
END_VAR
GetConfiguredPayloadSize := ServerConfiguration.PAYLOAD_STRING_SIZE;
END_METHOD

{attribute 'TcRpcEnable'}
METHOD PUBLIC HandleRequest : ResponseData;
VAR_INPUT
	SerializedHeader : STRING(ServerConfiguration.HEADER_STRING_SIZE);
	SerializedPayload : STRING(ServerConfiguration.PAYLOAD_STRING_SIZE);
END_VAR
VAR
	header : Header(SerializedHeader);
	request : Request(header, SerializedPayload);
	serverResponse : ServerResponse(headerAccessor);
END_VAR
middlewareStack.Handle(request, serverResponse);

IF NOT serverResponse.HeadersSent THEN
	serverResponse.Error('UNHANDLED_REQUEST', 'Unhandled Request');
END_IF

serverResponse.TryGetData(HandleRequest);
END_METHOD

METHOD PUBLIC RegisterApi
VAR_INPUT
	RpcApi : I_RpcApi;
END_VAR
RpcApi.RegisterSynchronousRpcHandlersWith(synchronousRpcHandlers);
RpcApi.RegisterAsynchronousRpcHandlersWith(asynchronousRpcHandlers);
registeredRpcApis.RegisterRpcApi(RpcApi);
END_METHOD

METHOD PUBLIC RegisterAsynchronousRpcHandler
VAR_INPUT
	MethodName : T_MAXSTRING;
	Handler : I_AsynchronousRpcHandler;
END_VAR
asynchronousRpcHandlers.RegisterHandler(MethodName, Handler);
END_METHOD

METHOD PUBLIC RegisterSynchronousRpcHandler
VAR_INPUT
	MethodName : T_MAXSTRING;
	Handler : I_SynchronousRpcHandler;
END_VAR
synchronousRpcHandlers.RegisterHandler(MethodName, Handler);
END_METHOD

PROPERTY PUBLIC SessionCount : DINT
GET
SessionCount := sessionManager.SessionCount;
END_GET
END_PROPERTY

METHOD PUBLIC Use
VAR_INPUT
	Middleware : I_Middleware;
END_VAR
middlewareStack.Use(Middleware);
END_METHOD

END_FUNCTION_BLOCK

// ---- mobject-server/_Internal/HeaderAccessor/HeaderAccessor.TcPOU
FUNCTION_BLOCK HeaderAccessor IMPLEMENTS I_SessionHeaderAccessor, I_ServerResponseHeaderAccessor, I_AsyncResponseHeaderAccessor, I_ChunkedResponseHeaderAccessor, I_ChunkedRequestsHeaderAccessor, I_RpcHeaderAccessor

PROPERTY PUBLIC ContentType_Json : T_MAXSTRING
GET
ContentType_Json := 'application/json';
END_GET
END_PROPERTY

PROPERTY PUBLIC HeaderKey_Accept : T_MAXSTRING
GET
HeaderKey_Accept := 'Accept';
END_GET
END_PROPERTY

PROPERTY PUBLIC HeaderKey_ChunkSequence : T_MAXSTRING
GET
HeaderKey_ChunkSequence := 'Chunk-Sequence';
END_GET
END_PROPERTY

PROPERTY PUBLIC HeaderKey_ChunkTotal : T_MAXSTRING
GET
HeaderKey_ChunkTotal := 'Chunk-Total';
END_GET
END_PROPERTY

PROPERTY PUBLIC HeaderKey_ContentType : T_MAXSTRING
GET
HeaderKey_ContentType := 'Content-Type';
END_GET
END_PROPERTY

PROPERTY PUBLIC HeaderKey_ErrorCode : T_MAXSTRING
GET
HeaderKey_ErrorCode := 'Error-Code';
END_GET
END_PROPERTY

PROPERTY PUBLIC HeaderKey_ErrorMessage : T_MAXSTRING
GET
HeaderKey_ErrorMessage := 'Error-Message';
END_GET
END_PROPERTY

PROPERTY PUBLIC HeaderKey_HasMoreChunks : T_MAXSTRING
GET
HeaderKey_HasMoreChunks := 'Has-More-Chunks';
END_GET
END_PROPERTY

PROPERTY PUBLIC HeaderKey_MethodName : T_MAXSTRING
GET
HeaderKey_MethodName := 'Method-Name';
END_GET
END_PROPERTY

PROPERTY PUBLIC HeaderKey_RequestId : T_MAXSTRING
GET
HeaderKey_RequestId := 'Request-Id';
END_GET
END_PROPERTY

PROPERTY PUBLIC HeaderKey_ResponseId : T_MAXSTRING
GET
HeaderKey_ResponseId := 'Response-Id';
END_GET
END_PROPERTY

PROPERTY PUBLIC HeaderKey_RetryDelay : T_MAXSTRING
GET
HeaderKey_RetryDelay := 'Retry-Delay';
END_GET
END_PROPERTY

PROPERTY PUBLIC HeaderKey_SessionId : T_MAXSTRING
GET
HeaderKey_SessionId := 'Session-Id';
END_GET
END_PROPERTY

PROPERTY PUBLIC HeaderKey_Status : T_MAXSTRING
GET
HeaderKey_Status := 'Status';
END_GET
END_PROPERTY

PROPERTY PUBLIC HeaderKey_Type : T_MAXSTRING
GET
HeaderKey_Type := 'Type';
END_GET
END_PROPERTY

PROPERTY PUBLIC StatusValue_Accepted : T_MAXSTRING
GET
StatusValue_Accepted := 'Accepted';
END_GET
END_PROPERTY

PROPERTY PUBLIC StatusValue_Busy : T_MAXSTRING
GET
StatusValue_Busy := 'Busy';
END_GET
END_PROPERTY

PROPERTY PUBLIC StatusValue_Error : T_MAXSTRING
GET
StatusValue_Error := 'Error';
END_GET
END_PROPERTY

PROPERTY PUBLIC StatusValue_Pending : T_MAXSTRING
GET
StatusValue_Pending := 'Pending';
END_GET
END_PROPERTY

PROPERTY PUBLIC StatusValue_Success : T_MAXSTRING
GET
StatusValue_Success := 'Success';
END_GET
END_PROPERTY

METHOD PUBLIC TryGetAcceptResponseFormatFromRequest : BOOL
VAR_INPUT
	Request : I_Request;
	Destination : ANY;
END_VAR
TryGetAcceptResponseFormatFromRequest := Request.Header.TryGetField(HeaderKey_Accept,Destination);
END_METHOD

METHOD PUBLIC TryGetChunkSequenceFromRequest : BOOL
VAR_INPUT
	Request : I_Request;
	Destination : REFERENCE TO DINT;
END_VAR
VAR
	chunkSequence : DINT;
END_VAR
IF NOT Request.Header.TryGetField(HeaderKey_ChunkSequence,chunkSequence) THEN
	RETURN;
END_IF

Destination := chunkSequence;
TryGetChunkSequenceFromRequest := TRUE;
END_METHOD

METHOD PUBLIC TryGetChunkTotalFromRequest : BOOL
VAR_INPUT
	Request : I_Request;
	Destination : REFERENCE TO DINT;
END_VAR
VAR
	chunkTotal : DINT;
END_VAR
IF NOT Request.Header.TryGetField(HeaderKey_ChunkTotal,chunkTotal) THEN
	RETURN;
END_IF

Destination := chunkTotal;
TryGetChunkTotalFromRequest := TRUE;
END_METHOD

METHOD PUBLIC TryGetContentTypeFromRequest : BOOL
VAR_INPUT
	Request : I_Request;
	Destination : ANY;
END_VAR
TryGetContentTypeFromRequest := Request.Header.TryGetField(HeaderKey_ContentType,Destination);
END_METHOD

METHOD PUBLIC TryGetHasMoreChunksFromRequest : BOOL
VAR_INPUT
	Request : I_Request;
	Destination : REFERENCE TO BOOL;
END_VAR
VAR
	hasMoreChunks : BOOL;
END_VAR
IF NOT Request.Header.TryGetField(HeaderKey_HasMoreChunks,hasMoreChunks) THEN
	RETURN;
END_IF

Destination := hasMoreChunks;
TryGetHasMoreChunksFromRequest := TRUE;
END_METHOD

METHOD PUBLIC TryGetMethodNameFromRequest : BOOL
VAR_INPUT
	Request : I_Request;
	Destination : ANY;
END_VAR
TryGetMethodNameFromRequest := Request.Header.TryGetField(HeaderKey_MethodName,Destination);
END_METHOD

METHOD PUBLIC TryGetRequestIdFromRequest : BOOL
VAR_INPUT
	Request : I_Request;
	Destination : REFERENCE TO T_MAXSTRING;
END_VAR
VAR
	requestId : T_MAXSTRING;
END_VAR
IF NOT Request.Header.TryGetField(HeaderKey_RequestId,requestId) THEN
	RETURN;
END_IF

Destination := requestId;
TryGetRequestIdFromRequest := TRUE;
END_METHOD

METHOD PUBLIC TryGetResponseIdFromRequest : BOOL
VAR_INPUT
	Request : I_Request;
	Destination : ANY;
END_VAR
TryGetResponseIdFromRequest := Request.Header.TryGetField(HeaderKey_ResponseId,Destination);
END_METHOD

METHOD PUBLIC TryGetSessionIdFromRequest : BOOL
VAR_INPUT
	Request : I_Request;
	Destination : REFERENCE TO T_MAXSTRING;
END_VAR
VAR
	sessionId : T_MAXSTRING;
END_VAR
IF NOT Request.Header.TryGetField(HeaderKey_SessionId, sessionId) THEN
	RETURN;
END_IF

Destination := sessionId;
TryGetSessionIdFromRequest := TRUE;
END_METHOD

METHOD PUBLIC TryGetSessionIdFromResponse : BOOL
VAR_INPUT
	Response : I_ServerResponse;
	Destination : ANY;
END_VAR
TryGetSessionIdFromResponse := Response.Header.TryGetField(HeaderKey_SessionId,Destination);
END_METHOD

METHOD PUBLIC TryGetTypeFromRequest : BOOL
VAR_INPUT
	Request : I_Request;
	Destination : ANY;
END_VAR
TryGetTypeFromRequest := Request.Header.TryGetField(HeaderKey_Type,Destination);
END_METHOD

METHOD PUBLIC UpdateRequestWithSessionId
VAR_INPUT
	Request : I_Request;
	SessionId : T_MAXSTRING;
END_VAR
Request.Header.TryWriteField(HeaderKey_SessionId,SessionId);
END_METHOD

METHOD PUBLIC UpdateResponseWithAccepted
VAR_INPUT
	Response : I_ServerResponse;
END_VAR
VAR
	status : T_MAXSTRING; // this was needed to fix the 4026 error with using ANY and properties
END_VAR
status := StatusValue_Accepted;
Response.Header.TryWriteField(HeaderKey_Status, status);
END_METHOD

METHOD PUBLIC UpdateResponseWithBusy
VAR_INPUT
	Response : I_ServerResponse;
END_VAR
VAR
	status : T_MAXSTRING; // this was needed to fix the 4026 error with using ANY and properties
END_VAR
status := StatusValue_Busy;
Response.Header.TryWriteField(HeaderKey_Status, status);
END_METHOD

METHOD PUBLIC UpdateResponseWithError
VAR_INPUT
	Response : I_ServerResponse;
	ErrorCode : T_MAXSTRING;
	Message : T_MAXSTRING;
END_VAR
VAR
	status : T_MAXSTRING; // this was needed to fix the 4026 error with using ANY and properties
END_VAR
status := StatusValue_Error;
Response.Header.TryWriteField(HeaderKey_Status, status);
Response.Header.TryWriteField(HeaderKey_ErrorCode, ErrorCode);
Response.Header.TryWriteField(HeaderKey_ErrorMessage, Message);
END_METHOD

METHOD PUBLIC UpdateResponseWithHasMoreChunks
VAR_INPUT
	Response : I_ServerResponse;
	ResponseId : T_MAXSTRING;
END_VAR
VAR
	hasMoreChunks : BOOL := TRUE;
END_VAR
Response.Header.TryWriteField(HeaderKey_ResponseId,ResponseId);
Response.Header.TryWriteField(HeaderKey_HasMoreChunks,hasMoreChunks);
END_METHOD

METHOD PUBLIC UpdateResponseWithPending
VAR_INPUT
	Response : I_ServerResponse;
	ResponseId : T_MAXSTRING;
	RetryDelayInMs : UDINT;
END_VAR
VAR
	retryDelayInMsString : T_MAXSTRING;
	status : T_MAXSTRING; // this was needed to fix the 4026 error with using ANY and properties
END_VAR
status := StatusValue_Pending;
Response.Header.TryWriteField(HeaderKey_Status, status);
Response.Header.TryWriteField(HeaderKey_ResponseId, ResponseId);

IF RetryDelayInMs > 0 THEN
	retryDelayInMsString := UDINT_TO_STRING(RetryDelayInMs);
	Response.Header.TryWriteField(HeaderKey_RetryDelay, retryDelayInMsString);
END_IF
END_METHOD

METHOD PUBLIC UpdateResponseWithSessionId
VAR_INPUT
	Response : I_ServerResponse;
	SessionId : T_MAXSTRING;
END_VAR
Response.Header.TryWriteField(HeaderKey_SessionId,SessionId);
END_METHOD

METHOD PUBLIC UpdateResponseWithSuccess
VAR_INPUT
	Response : I_ServerResponse;
END_VAR
VAR
	status : T_MAXSTRING; // this was needed to fix the 4026 error with using ANY and properties
END_VAR
status := StatusValue_Success;
Response.Header.TryWriteField(HeaderKey_Status, status);
END_METHOD

END_FUNCTION_BLOCK

// ---- mobject-server/_Internal/Request/Request.TcPOU
{attribute 'linkalways'} 
{attribute 'no_explicit_call' := 'This FB is a CLASS and must be accessed using methods or properties'}
{attribute 'enable_dynamic_creation'}
FUNCTION_BLOCK Request Extends Disposable IMPLEMENTS I_Request
VAR
	_header : I_Header;
	_payloadAddress : POINTER TO STRING(0);
	_payloadSizeInBytes : UDINT;	
	_createdTimestamp : SystemTimestamp;
END_VAR

PROPERTY PUBLIC CreatedTimestamp : I_Timestamp
GET
CreatedTimestamp := _createdTimestamp;
END_GET
END_PROPERTY

METHOD FB_init : BOOL
VAR_INPUT
	bInitRetains : BOOL; // if TRUE, the retain variables are initialized (warm start / cold start)
	bInCopyCode : BOOL;  // if TRUE, the instance afterwards gets moved into the copy code (online change)
	Header : I_Header;
	Payload : ANY_STRING;
END_VAR
_header := Header;
_payloadSizeInBytes := DINT_TO_UDINT(Payload.diSize);
_payloadAddress := Payload.pValue;
END_METHOD

PROPERTY PUBLIC Header : I_Header
GET
Header := _header;
END_GET
END_PROPERTY

PROPERTY PUBLIC PayloadAddress : POINTER TO STRING
GET
PayloadAddress := _payloadAddress;
END_GET
END_PROPERTY

PROPERTY PUBLIC PayloadSizeInBytes : UDINT
GET
PayloadSizeInBytes := _payloadSizeInBytes;
END_GET
END_PROPERTY

END_FUNCTION_BLOCK

// ---- mobject-server/_Internal/TimeStamp/SystemTimestamp.TcPOU
FUNCTION_BLOCK SystemTimestamp Implements I_Timestamp
VAR
	recordedTime : ULINT;
END_VAR

METHOD FB_init : BOOL
VAR_INPUT
	bInitRetains : BOOL; // if TRUE, the retain variables are initialized (warm start / cold start)
	bInCopyCode : BOOL;  // if TRUE, the instance afterwards gets moved into the copy code (online change)
END_VAR
SetNow();
END_METHOD

METHOD PUBLIC IsDurationElapsed : BOOL
VAR_INPUT
	Duration : TIME;
END_VAR
VAR
	currentTime : ULINT;
	elapsedDuration : ULINT;
	durationInHundredNs : ULINT;
END_VAR
currentTime := F_GetSystemTime();

// Convert duration from milliseconds to 100-nanosecond intervals.
// Since 1 ms = 10,000 * 100 ns.
durationInHundredNs := TIME_TO_ULINT(duration) * 10000; 

// Calculate the time that must elapse before the timestamp is considered 'expired'.
elapsedDuration := recordedTime + durationInHundredNs;

// Check if the current time is beyond the elapsed duration.
IsDurationElapsed := currentTime > elapsedDuration;
END_METHOD

METHOD PUBLIC SetNow
VAR_INPUT
END_VAR
recordedTime := F_GetSystemTime();
END_METHOD

PROPERTY PUBLIC TimeSince : TIME
GET
VAR
	currentTime : ULINT;
	elapsedDurationInHundredNs : ULINT;
	convertTime : ULINT;
END_VAR
currentTime := F_GetSystemTime();

elapsedDurationInHundredNs := currentTime - recordedTime;
convertTime := elapsedDurationInHundredNs / 10000;
TimeSince := ULINT_TO_TIME(convertTime);
END_GET
END_PROPERTY

END_FUNCTION_BLOCK

// ---- mobject-server/_Internal/Header/Header.TcPOU
{attribute 'linkalways'} 
{attribute 'no_explicit_call' := 'This FB is a CLASS and must be accessed using methods or properties'}
{attribute 'enable_dynamic_creation'}
FUNCTION_BLOCK Header IMPLEMENTS I_Header
VAR
	jsonParser : JsonDomParser;
END_VAR

METHOD FB_exit : BOOL
VAR_INPUT
	bInCopyCode : BOOL; // if TRUE, the exit method is called for exiting an instance that is copied afterwards (online change).
END_VAR
IF bInCopyCode THEN
	RETURN;
END_IF

jsonParser.NewDocument();
END_METHOD

METHOD FB_init : BOOL
VAR_INPUT
	bInitRetains : BOOL; // if TRUE, the retain variables are initialized (warm start / cold start)
	bInCopyCode : BOOL;  // if TRUE, the instance afterwards gets moved into the copy code (online change)
	InitialHeader : REFERENCE TO STRING(ServerConfiguration.HEADER_STRING_SIZE);
END_VAR
VAR
	root : SJsonValue;
END_VAR
IF __ISVALIDREF(InitialHeader) THEN
	root := jsonParser.ParseDocument(InitialHeader);
ELSE
	root := jsonParser.NewDocument();
	jsonParser.SetObject(root);
END_IF
END_METHOD

METHOD PUBLIC ToString
VAR_INPUT
	Destination : REFERENCE TO STRING(ServerConfiguration.HEADER_STRING_SIZE);
END_VAR
jsonParser.CopyDocument(Destination,sizeof(Destination));
END_METHOD

METHOD PUBLIC TryGetField : BOOL;
VAR_INPUT
	Key : STRING;
	Destination : ANY;
END_VAR
IF Key = '' THEN
	RETURN;
END_IF

TryGetField := jsonParser.TryRead(Key, Destination);
END_METHOD

METHOD PUBLIC TryWriteField : BOOL;
VAR_INPUT
	Key : STRING;
	Source : ANY;
END_VAR
IF Key = '' THEN
	RETURN;
END_IF

TryWriteField := jsonParser.TryWrite(Key, Source);
END_METHOD

END_FUNCTION_BLOCK

// ---- mobject-server/_Internal/Sessions/Session/Session.TcPOU
{attribute 'linkalways'} 
{attribute 'no_explicit_call' := 'This FB is a CLASS and must be accessed using methods or properties'}
{attribute 'enable_dynamic_creation'}
FUNCTION_BLOCK Session EXTENDS Disposable IMPLEMENTS I_Session
VAR
	_id : T_MAXSTRING;
	_lastAccessedTimestamp : SystemTimestamp;
	sessionStorage : Dictionary;
END_VAR

METHOD PUBLIC AddOrUpdateStorage
VAR_INPUT
	StorageId : T_MAXSTRING;
	Source : I_SessionData;
END_VAR
sessionStorage.AddOrUpdate(StorageId, Source);
END_METHOD

METHOD PUBLIC DisposeAllDataFromStorage
VAR_INPUT
END_VAR
VAR
	enumerator : I_ForwardEnumerator;
	sessionData : I_SessionData;
END_VAR
enumerator := sessionStorage.GetEnumerator();

WHILE enumerator.MoveNext() DO
	IF enumerator.TryGet(sessionData) THEN
		sessionData.Dispose();
	END_IF
END_WHILE

enumerator.Dispose();
sessionStorage.Clear();
END_METHOD

METHOD PUBLIC DisposeDataFromStorage
VAR_INPUT
	StorageId : T_MAXSTRING;
END_VAR
VAR
	sessionData : I_SessionData;
END_VAR
IF NOT sessionStorage.TryGetValue(StorageId,sessionData) THEN
	RETURN;
END_IF

sessionData.Dispose();
sessionStorage.Remove(StorageId);
END_METHOD

METHOD FB_exit : BOOL
VAR_INPUT
	bInCopyCode : BOOL; // if TRUE, the exit method is called for exiting an instance that is copied afterwards (online change).
END_VAR
IF bInCopyCode THEN
	RETURN;
END_IF

DisposeAllDataFromStorage();
END_METHOD

METHOD FB_init : BOOL
VAR_INPUT
	bInitRetains : BOOL; // if TRUE, the retain variables are initialized (warm start / cold start)
	bInCopyCode : BOOL;  // if TRUE, the instance afterwards gets moved into the copy code (online change)
	SessionId : T_MAXSTRING;
END_VAR
_id := SessionId;
END_METHOD

PROPERTY PUBLIC Id : T_MAXSTRING
GET
Id := _id;
END_GET
END_PROPERTY

PROPERTY PUBLIC LastAccessedTimestamp : I_TimeStamp
GET
LastAccessedTimestamp := _lastAccessedTimestamp;
END_GET
END_PROPERTY

METHOD PUBLIC Refresh
VAR_INPUT
END_VAR
_lastAccessedTimestamp.SetNow();
END_METHOD

METHOD PUBLIC TryGetDataFromStorage : BOOL
VAR_INPUT
	StorageId : T_MAXSTRING;
	Destination : REFERENCE TO I_SessionData;
END_VAR
TryGetDataFromStorage := sessionStorage.TryGetValue(StorageId, Destination);
END_METHOD

END_FUNCTION_BLOCK

// ---- mobject-server/_Internal/Middleware/Stack/MiddlewareStack.TcPOU
{attribute 'linkalways'} 
{attribute 'no_explicit_call' := 'This FB is a CLASS and must be accessed using methods or properties'}
{attribute 'enable_dynamic_creation'}
FUNCTION_BLOCK MiddlewareStack
VAR
	InitialHandler : I_Middleware;
END_VAR

METHOD PUBLIC Handle
VAR_INPUT
	Request : I_Request;
	Response : I_ServerResponse;
END_VAR
IF initialHandler = 0 THEN
	RETURN;
END_IF

initialHandler.Handle(Request, Response);
END_METHOD

METHOD PUBLIC Use
VAR_INPUT
	Handler : I_Middleware;
END_VAR
VAR
	currentHandler : I_Middleware;
END_VAR;
IF initialHandler = 0 THEN
	initialHandler := Handler;
	RETURN;
END_IF

currentHandler := InitialHandler;

WHILE currentHandler.NextMiddleware <> 0 DO
	currentHandler := currentHandler.NextMiddleware;
END_WHILE

currentHandler.NextMiddleware := Handler;
END_METHOD

END_FUNCTION_BLOCK

// ---- mobject-server/_Internal/ResponseId/SequentialResponseIdGenerator.TcPOU
{attribute 'linkalways'} 
{attribute 'no_explicit_call' := 'This FB is a CLASS and must be accessed using methods or properties'}
{attribute 'enable_dynamic_creation'}
FUNCTION_BLOCK SequentialResponseIdGenerator IMPLEMENTS I_ResponseIdGenerator
VAR
	currentCount : UDINT;
END_VAR

METHOD PUBLIC Generate : T_MAXSTRING
VAR_INPUT
END_VAR
currentCount := currentCount + 1;
Generate := UDINT_TO_STRING(currentCount);
END_METHOD

END_FUNCTION_BLOCK

// ---- mobject-server/_Internal/Sessions/SessionId/SequentialSessionIdGenerator.TcPOU
{attribute 'linkalways'} 
{attribute 'no_explicit_call' := 'This FB is a CLASS and must be accessed using methods or properties'}
{attribute 'enable_dynamic_creation'}
FUNCTION_BLOCK SequentialSessionIdGenerator Implements I_SessionIdGenerator
VAR
	currentCount : UDINT;
END_VAR

METHOD PUBLIC Generate : T_MAXSTRING
VAR_INPUT
END_VAR
currentCount := currentCount + 1;
Generate := UDINT_TO_STRING(currentCount);
END_METHOD

END_FUNCTION_BLOCK

// ---- mobject-server/_Internal/Sessions/Manager/SessionManager.TcPOU
{attribute 'linkalways'} 
{attribute 'no_explicit_call' := 'This FB is a CLASS and must be accessed using methods or properties'}
{attribute 'enable_dynamic_creation'}
FUNCTION_BLOCK SessionManager implements I_SessionManager, I_SessionStorage
VAR
	activeSessions : Dictionary;
	sessionIdGenerator : I_SessionIdGenerator;
	currentStorageId : UDINT;
	sessionMaxLife : TIME;
END_VAR

METHOD PUBLIC CheckForExpiredSessions
VAR_INPUT
END_VAR
VAR
	enumerator : I_ForwardEnumerator;
	session : I_Session;
	expiredSessions : Stack;
END_VAR
enumerator := activeSessions.GetEnumerator();

WHILE enumerator.MoveNext() DO
	IF enumerator.TryGet(session) THEN
		IF session.LastAccessedTimestamp.IsDurationElapsed(sessionMaxLife) THEN
			expiredSessions.Push(session);
		END_IF
	END_IF
END_WHILE

enumerator.Dispose();

WHILE expiredSessions.TryPop(session) DO
	DisposeSession(session.Id);
END_WHILE
END_METHOD

METHOD PRIVATE CreateNewSession : I_Session
VAR
	id : T_MAXSTRING;
	pSession : POINTER TO Session;
END_VAR
id := sessionIdGenerator.Generate();
pSession := __NEW(Session(SessionId := id));
CreateNewSession := pSession^;
END_METHOD

METHOD PUBLIC CreateSession : T_MAXSTRING;
VAR
	session : I_Session;
END_VAR
session := CreateNewSession();
activeSessions.AddOrUpdate(session.Id, session);
CreateSession := session.Id;
END_METHOD

METHOD PUBLIC CyclicCall
VAR_INPUT
END_VAR
CheckForExpiredSessions();
END_METHOD

METHOD PUBLIC DisposeAllSessions
VAR_INPUT
END_VAR
VAR
	enumerator : I_ForwardEnumerator;
	session : I_Session;
END_VAR
enumerator := activeSessions.GetEnumerator();

WHILE enumerator.MoveNext() DO
	if enumerator.TryGet(session) then
		session.Dispose();
	END_IF
END_WHILE

enumerator.Dispose();
activeSessions.Clear();
END_METHOD

METHOD PUBLIC DisposeSession
VAR_INPUT
	Id : T_MAXSTRING;
END_VAR
VAR
	session : I_Session;
END_VAR
IF NOT activeSessions.TryGetValue(Id, session) THEN
	RETURN;
END_IF

session.Dispose();
activeSessions.Remove(Id);
END_METHOD

METHOD PUBLIC DisposeSessionDataById
VAR_INPUT
	SessionId : T_MAXSTRING;
	StorageId : T_MAXSTRING;
END_VAR
VAR
	session : I_Session;
	sessionData : I_SessionData;
END_VAR
IF StorageId = '' THEN 
	RETURN;
END_IF

IF NOT activeSessions.TryGetValue(SessionId, session) THEN
	RETURN;
END_IF

IF NOT session.TryGetDataFromStorage(StorageId, sessionData) THEN
	RETURN;
END_IF

session.DisposeDataFromStorage(StorageId);
END_METHOD

METHOD FB_exit : BOOL
VAR_INPUT
	bInCopyCode : BOOL; // if TRUE, the exit method is called for exiting an instance that is copied afterwards (online change).
END_VAR
IF bInCopyCode THEN
	RETURN;
END_IF

DisposeAllSessions();
END_METHOD

METHOD FB_init : BOOL
VAR_INPUT
	bInitRetains : BOOL; // if TRUE, the retain variables are initialized (warm start / cold start)
	bInCopyCode : BOOL;  // if TRUE, the instance afterwards gets moved into the copy code (online change)
	SessionIdGenerator : I_SessionIdGenerator;
	SessionMaxLife : TIME;
END_VAR
THIS^.sessionIdGenerator := SessionIdGenerator;
THIS^.sessionMaxLife := SessionMaxLife;
END_METHOD

METHOD PUBLIC IsValidSession : BOOL
VAR_INPUT
	Id : T_MAXSTRING;
END_VAR
IsValidSession := activeSessions.ContainsKey(Id);
END_METHOD

METHOD PUBLIC RefreshSession
VAR_INPUT
	Id : T_MAXSTRING;
END_VAR
VAR
	session : I_Session;
END_VAR
IF NOT activeSessions.TryGetValue(Id, session) THEN
	RETURN;
END_IF

session.Refresh();
END_METHOD

PROPERTY PUBLIC SessionCount : DINT
GET
SessionCount := activeSessions.Count;
END_GET
END_PROPERTY

METHOD PUBLIC TryRetrieveSessionDataById : BOOL
VAR_INPUT
	SessionId : T_MAXSTRING;
	StorageId : T_MAXSTRING;
	Destination : REFERENCE TO I_SessionData;
END_VAR
VAR
	session : I_Session;
END_VAR
IF NOT activeSessions.TryGetValue(SessionId, session) THEN
	RETURN;
END_IF

TryRetrieveSessionDataById := session.TryGetDataFromStorage(StorageId, Destination);
END_METHOD

METHOD PUBLIC TryStoreSessionDataById : BOOL
VAR_INPUT
	SessionId : T_MAXSTRING;
	StorageId : T_MAXSTRING;
	Source : I_SessionData;
END_VAR
VAR
	session : I_Session;
END_VAR
IF StorageId = '' THEN 
	RETURN;
END_IF

IF NOT activeSessions.TryGetValue(SessionId, session) THEN
	RETURN;
END_IF

session.AddOrUpdateStorage(StorageId, Source);
TryStoreSessionDataById := TRUE;
END_METHOD

END_FUNCTION_BLOCK

// ---- mobject-server/_Internal/Sessions/Middleware/SessionsMiddleware.TcPOU
{attribute 'linkalways'} 
{attribute 'no_explicit_call' := 'This FB is a CLASS and must be accessed using methods or properties'}
{attribute 'enable_dynamic_creation'}
FUNCTION_BLOCK SessionsMiddleware EXTENDS MiddlewareBase
VAR
	sessionManager: I_SessionManager;
	headerAccessor : I_SessionHeaderAccessor;
END_VAR

METHOD FB_init : BOOL
VAR_INPUT
	bInitRetains : BOOL; // if TRUE, the retain variables are initialized (warm start / cold start)
	bInCopyCode : BOOL;  // if TRUE, the instance afterwards gets moved into the copy code (online change)
	SessionManager : I_SessionManager;
	HeaderAccessor : I_SessionHeaderAccessor;
END_VAR
THIS^.sessionManager := SessionManager;
THIS^.headerAccessor := HeaderAccessor;
END_METHOD

METHOD PUBLIC Handle
VAR_INPUT
	Request : I_Request;
	Response : I_ServerResponse;
END_VAR
VAR
	sessionId : T_MAXSTRING;
	responseId : T_MAXSTRING;
END_VAR
IF (NOT headerAccessor.TryGetSessionIdFromRequest(Request, sessionId)) OR_ELSE (NOT sessionManager.IsValidSession(sessionId)) THEN

	IF headerAccessor.TryGetResponseIdFromRequest(Request, responseId) THEN
		Response.Error(
			'SESSION_EXPIRED',
			'The session for this follow-up has expired. The original request outcome is unknown.'
		);
		RETURN;
	END_IF

	sessionId := sessionManager.CreateSession();
	headerAccessor.UpdateRequestWithSessionId(Request,sessionId);
END_IF

sessionManager.RefreshSession(sessionId);

headerAccessor.UpdateResponseWithSessionId(Response, sessionId);
Next(Request, Response);
END_METHOD

END_FUNCTION_BLOCK

// ---- mobject-server/_Internal/Middleware/Base/MiddlewareBase.TcPOU
{attribute 'linkalways'} 
{attribute 'no_explicit_call' := 'This FB is a CLASS and must be accessed using methods or properties'}
{attribute 'enable_dynamic_creation'}
FUNCTION_BLOCK ABSTRACT MiddlewareBase implements I_Middleware
VAR
	_next : I_Middleware;
END_VAR

METHOD PUBLIC ABSTRACT Handle
VAR_INPUT
	Request : I_Request;
	Response : I_ServerResponse;
END_VAR
// Call next to pass the request and response to the next handler
// Next(Request, Response);
END_METHOD

METHOD PROTECTED Next
VAR_INPUT
	Request : I_Request;
	Response : I_ServerResponse;
END_VAR
IF _next = 0 THEN
	RETURN;
END_IF

_next.Handle(Request, Response);
END_METHOD

PROPERTY PUBLIC NextMiddleware : I_Middleware
GET
NextMiddleware := _next;
END_GET
SET
_next := NextMiddleware;
END_SET
END_PROPERTY

END_FUNCTION_BLOCK

// ---- mobject-server/_Internal/ChunkedRequests/Manager/ChunkedRequestsManager.TcPOU
{attribute 'linkalways'} 
{attribute 'no_explicit_call' := 'This FB is a CLASS and must be accessed using methods or properties'}
{attribute 'enable_dynamic_creation'}
FUNCTION_BLOCK ChunkedRequestsManager IMPLEMENTS I_ChunkedRequestsManager
VAR
	maximumChunkSizeInBytes : UDINT;
	sessionStorage : I_SessionStorage;
	headerAccessor : I_ChunkedRequestsHeaderAccessor;
END_VAR

METHOD PRIVATE CreateChunkedRequestData : I_ChunkedRequestData
VAR_INPUT
	RequestChunkSizeInBytes : UDINT;
	RequestChunkCount : UDINT;
END_VAR
VAR
	pChunkedRequestData : POINTER TO ChunkedRequestData;
END_VAR
pChunkedRequestData := __NEW(ChunkedRequestData(ChunkSizeInBytes := RequestChunkSizeInBytes, ChunkCount := RequestChunkCount));
CreateChunkedRequestData := pChunkedRequestData^;
END_METHOD

METHOD FB_init : BOOL
VAR_INPUT
	bInitRetains : BOOL; // if TRUE, the retain variables are initialized (warm start / cold start)
	bInCopyCode : BOOL;  // if TRUE, the instance afterwards gets moved into the copy code (online change)
	MaximumChunkSizeInBytes : UDINT;
	SessionStorage : I_SessionStorage;
	HeaderAccessor : I_ChunkedRequestsHeaderAccessor;
END_VAR
THIS^.maximumChunkSizeInBytes := MaximumChunkSizeInBytes;
THIS^.sessionStorage := SessionStorage;
THIS^.headerAccessor := HeaderAccessor;
END_METHOD

METHOD PUBLIC TryHandleIncomingRequest : BOOL
VAR_INPUT
	Request : I_Request;
	Response : I_ServerResponse;
	NextMidleware : I_Middleware;
END_VAR
VAR 
	hasChunkSequenceHeader : BOOL;
	chunkSequence : DINT;
	hasChunkTotalHeader : BOOL;
	chunkTotal : DINT;
	hasMoreChunksHeader : BOOL;
	hasMoreChunks : BOOL;
	requestId : T_MAXSTRING;
	sessionId : T_MAXSTRING;
	sessionData : I_SessionData;
	chunkedRequestData : I_ChunkedRequestData;
	chunkedRequest : ChunkedRequest(Request, chunkedRequestData);
END_VAR
hasChunkSequenceHeader := headerAccessor.TryGetChunkSequenceFromRequest(Request, chunkSequence);
hasChunkTotalHeader := headerAccessor.TryGetChunkTotalFromRequest(Request, chunkTotal);
hasMoreChunksHeader := headerAccessor.TryGetHasMoreChunksFromRequest(Request, hasMoreChunks);

IF (NOT hasChunkSequenceHeader) AND (NOT hasChunkTotalHeader) AND (NOT hasMoreChunksHeader) THEN
	// this is not a chunked request, simply return and it will be handled by the next middleware automatically.
	RETURN;
END_IF

// when reaching here we know that the request has at least one of the headers associated with chunked requests
// from this point on, we simply validate until we know we have all the required parts. 

IF NOT hasChunkSequenceHeader THEN
	response.Error('INVALID_CHUNK_HEADER','Chunked Request found, but chunk sequence header data is missing');
	TryHandleIncomingRequest := TRUE;
	RETURN;
END_IF

IF chunkSequence = 0 THEN
	response.Error('INVALID_CHUNK_HEADER','Chunk sequence 0 received, chunks must start from 1');
	TryHandleIncomingRequest := TRUE;
	RETURN;
END_IF

IF NOT hasChunkTotalHeader THEN
	response.Error('INVALID_CHUNK_HEADER','Chunked Request found, but chunk total header data is missing');
	TryHandleIncomingRequest := TRUE;
	RETURN;
END_IF

IF chunkSequence > chunkTotal THEN
	response.Error('INVALID_CHUNK_HEADER','Chunk sequence is greater than the chunk total');
	TryHandleIncomingRequest := TRUE;
	RETURN;
END_IF

IF NOT hasMoreChunksHeader THEN
	response.Error('INVALID_CHUNK_HEADER','Chunked Request found, but has more chunks header data is missing');
	TryHandleIncomingRequest := TRUE;
	RETURN;
END_IF

IF NOT headerAccessor.TryGetRequestIdFromRequest(Request, requestId) THEN
	response.Error('INVALID_CHUNK_HEADER','Chunked Request found, but request id header data is missing');
	TryHandleIncomingRequest := TRUE;
	RETURN;
END_IF

IF NOT headerAccessor.TryGetSessionIdFromRequest(Request, sessionId) THEN
	response.Error('INVALID_CHUNK_HEADER','Chunked Request found, but session id header data is missing');
	TryHandleIncomingRequest := TRUE;
	RETURN;
END_IF

// at this point we know we have all of the data required for handling a chunked request

IF NOT sessionStorage.TryRetrieveSessionDataById(sessionId, requestId, sessionData) THEN

	// Nothing stored for a chunk which is not the first means the earlier chunks
	// have gone - the session holding them expired or was replaced part way
	// through the upload.  Opening a fresh buffer here would quietly discard
	// them and leave a request which can never reach its chunk total, so the
	// client would wait until it timed out with no idea why.  Fail it instead so
	// the whole request can be sent again.
	IF chunkSequence > 1 THEN
		response.Error('CHUNKED_REQUEST_LOST', 'The earlier chunks of this request are no longer held by the server. The request must be sent again from the first chunk.');
		TryHandleIncomingRequest := TRUE;
		RETURN;
	END_IF

	chunkedRequestData := CreateChunkedRequestData(maximumChunkSizeInBytes, DINT_TO_UDINT(chunkTotal));
	sessionStorage.TryStoreSessionDataById(sessionId, requestId, chunkedRequestData);
ELSIF NOT __QUERYINTERFACE(sessionData, chunkedRequestData) THEN
	response.Error('SERVER_INTERNAL_ERROR','Server was unable to retreive previous session data as chunked request data');
	TryHandleIncomingRequest := TRUE;
	RETURN;
END_IF

IF NOT chunkedRequestData.TryAddChunkedPayload(request.PayloadAddress, request.PayloadSizeInBytes, chunkSequence) THEN
	response.Error('SERVER_INTERNAL_ERROR','Unable to store request payload in chunk session storage');
	sessionStorage.DisposeSessionDataById(sessionId, requestId);
	TryHandleIncomingRequest := TRUE;
	RETURN;
END_IF

IF NOT chunkedRequestData.IsComplete THEN
	Response.Accepted();
	TryHandleIncomingRequest := TRUE;
	RETURN;
END_IF

NextMidleware.Handle(chunkedRequest, Response);
sessionStorage.DisposeSessionDataById(sessionId, requestId);
TryHandleIncomingRequest := TRUE;
END_METHOD

END_FUNCTION_BLOCK

// ---- mobject-server/_Internal/ChunkedRequests/SessionData/ChunkedRequestData.TcPOU
{attribute 'linkalways'} 
{attribute 'no_explicit_call' := 'This FB is a CLASS and must be accessed using methods or properties'}
{attribute 'enable_dynamic_creation'}
FUNCTION_BLOCK ChunkedRequestData EXTENDS Disposable IMPLEMENTS I_ChunkedRequestData
VAR
	maximumChunkSizeInBytes : UDINT;
	totalReceivedChunks : UDINT;
	totalExpectedChunks : UDINT;
	pPayloadBuffer : POINTER TO STRING;
	payloadBufferSize : UDINT;
END_VAR

METHOD PRIVATE CreateBuffer
VAR_INPUT
	SizeInBytes : UDINT;
END_VAR
payloadBufferSize := SizeInBytes;
pPayloadBuffer := __NEW(BYTE, SizeInBytes);
memset(pPayloadBuffer, 0, SizeInBytes);
END_METHOD

METHOD PRIVATE DestroyBuffer
VAR_INPUT
END_VAR
IF pPayloadBuffer = 0 THEN
	RETURN;
END_IF

__DELETE(pPayloadBuffer);
pPayloadBuffer := 0;
END_METHOD

METHOD FB_exit : BOOL
VAR_INPUT
	bInCopyCode : BOOL; // if TRUE, the exit method is called for exiting an instance that is copied afterwards (online change).
END_VAR
IF bInCopyCode THEN
	RETURN;
END_IF

DestroyBuffer();
END_METHOD

METHOD FB_init : BOOL
VAR_INPUT
	bInitRetains : BOOL; // if TRUE, the retain variables are initialized (warm start / cold start)
	bInCopyCode : BOOL;  // if TRUE, the instance afterwards gets moved into the copy code (online change)
	ChunkSizeInBytes : UDINT;
	ChunkCount : UDINT;
END_VAR
maximumChunkSizeInBytes := ChunkSizeInBytes;
totalExpectedChunks := ChunkCount;
CreateBuffer(ChunkSizeInBytes * ChunkCount);
END_METHOD

PROPERTY PUBLIC IsComplete : BOOL
GET
IsComplete := totalReceivedChunks = totalExpectedChunks;
END_GET
END_PROPERTY

PROPERTY PUBLIC PayloadAddress : POINTER TO STRING
GET
PayloadAddress := pPayloadBuffer;
END_GET
END_PROPERTY

PROPERTY PUBLIC PayloadSizeInBytes : UDINT
GET
PayloadSizeInBytes := payloadBufferSize;
END_GET
END_PROPERTY

METHOD PUBLIC TryAddChunkedPayload : BOOL;
VAR_INPUT
	PayloadAddress : POINTER TO STRING;
	PayloadSize : UDINT;
	ChunkSequence : DINT;
END_VAR
VAR
	offset : UDINT;
	pBufferChunkLocation : POINTER TO BYTE;
END_VAR
IF totalReceivedChunks >= totalExpectedChunks THEN
	RETURN;
END_IF

IF PayloadSize > maximumChunkSizeInBytes THEN
	RETURN;
END_IF

// The payload is appended in arrival order rather than placed by index, so a
// chunk which is not the one due next cannot be stored correctly.  Rejecting it
// turns what would otherwise be silent corruption of the assembled request into
// a clean failure.  This covers a duplicate too, which would otherwise be
// appended twice and counted towards completion twice.
IF ChunkSequence <> UDINT_TO_DINT(totalReceivedChunks) + 1 THEN
	RETURN;
END_IF

concat2(pPayloadBuffer, PayloadAddress, pPayloadBuffer, payloadBufferSize);
totalReceivedChunks := totalReceivedChunks + 1;

TryAddChunkedPayload := TRUE;
END_METHOD

END_FUNCTION_BLOCK

// ---- mobject-server/_Internal/ChunkedRequests/ChunkedRequest/ChunkedRequest.TcPOU
{attribute 'linkalways'} 
{attribute 'no_explicit_call' := 'This FB is a CLASS and must be accessed using methods or properties'}
{attribute 'enable_dynamic_creation'}
FUNCTION_BLOCK ChunkedRequest EXTENDS Disposable IMPLEMENTS I_Request
VAR
	request : I_Request;
	chunkedRequestData : REFERENCE TO I_ChunkedRequestData;
END_VAR

PROPERTY PUBLIC CreatedTimestamp : I_Timestamp
GET
CreatedTimestamp := request.CreatedTimestamp;
END_GET
END_PROPERTY

METHOD FB_init : BOOL
VAR_INPUT
	bInitRetains : BOOL; // if TRUE, the retain variables are initialized (warm start / cold start)
	bInCopyCode : BOOL;  // if TRUE, the instance afterwards gets moved into the copy code (online change)
	Request : I_Request;
	ChunkedRequestData : Reference to I_ChunkedRequestData;
END_VAR
THIS^.request := Request;
THIS^.chunkedRequestData REF= ChunkedRequestData;
END_METHOD

PROPERTY PUBLIC Header : I_Header
GET
Header := request.Header;
END_GET
END_PROPERTY

PROPERTY PUBLIC PayloadAddress : POINTER TO STRING
GET
IF chunkedRequestData = 0 THEN
	RETURN;
END_IF

PayloadAddress := chunkedRequestData.PayloadAddress;
END_GET
END_PROPERTY

PROPERTY PUBLIC PayloadSizeInBytes : UDINT
GET
IF chunkedRequestData = 0 THEN
	RETURN;
END_IF

PayloadSizeInBytes := chunkedRequestData.PayloadSizeInBytes;
END_GET
END_PROPERTY

END_FUNCTION_BLOCK

// ---- mobject-server/_Internal/ChunkedRequests/Middleware/ChunkedRequestsMiddleware.TcPOU
{attribute 'linkalways'} 
{attribute 'no_explicit_call' := 'This FB is a CLASS and must be accessed using methods or properties'}
{attribute 'enable_dynamic_creation'}
FUNCTION_BLOCK ChunkedRequestsMiddleware EXTENDS MiddlewareBase
VAR
	chunkedRequestsManager : I_ChunkedRequestsManager;
END_VAR

METHOD FB_init : BOOL
VAR_INPUT
	bInitRetains : BOOL; // if TRUE, the retain variables are initialized (warm start / cold start)
	bInCopyCode : BOOL;  // if TRUE, the instance afterwards gets moved into the copy code (online change)
	ChunkedRequestsManager : I_ChunkedRequestsManager;
END_VAR
THIS^.chunkedRequestsManager := ChunkedRequestsManager;
END_METHOD

METHOD PUBLIC Handle
VAR_INPUT
	Request : I_Request;
	Response : I_ServerResponse;
END_VAR
VAR
	hasMoreChunks : BOOL;
END_VAR
IF chunkedRequestsManager.TryHandleIncomingRequest(Request, Response, NextMiddleware) THEN
	RETURN;
END_IF

Next(Request, Response);
END_METHOD

END_FUNCTION_BLOCK

// ---- mobject-server/_Internal/ChunkedResponses/Manager/ChunkedResponseManager.TcPOU
{attribute 'linkalways'} 
{attribute 'no_explicit_call' := 'This FB is a CLASS and must be accessed using methods or properties'}
{attribute 'enable_dynamic_creation'}
FUNCTION_BLOCK ChunkedResponseManager IMPLEMENTS I_ChunkedResponseManager
VAR
	// buffer size including the null terminator
	maximumChunkSizeInBytes : UDINT;
	// data bytes actually transmittable per chunk.  SendNextChunk reserves the last
	// byte for the null terminator, so this is always one less than the buffer size.
	maximumPayloadBytesPerChunk : UDINT;
	sessionStorage : I_SessionStorage;
	responseIdGenerator : I_ResponseIdGenerator;
	headerAccessor : I_ChunkedResponseHeaderAccessor;
END_VAR

METHOD PUBLIC CreateChunkedResponseData : I_ChunkedResponseData
VAR_INPUT
	DataAddress : PVOID;
	DataSize : UDINT;
END_VAR
VAR
	pChunkedResponseData : POINTER TO ChunkedResponseData;
END_VAR
pChunkedResponseData := __NEW(ChunkedResponseData(Address := DataAddress, Size:=DataSize));
CreateChunkedResponseData := pChunkedResponseData^;
END_METHOD

METHOD FB_init : BOOL
VAR_INPUT
	bInitRetains : BOOL; // if TRUE, the retain variables are initialized (warm start / cold start)
	bInCopyCode : BOOL;  // if TRUE, the instance afterwards gets moved into the copy code (online change)
	MaximumChunkSizeInBytes : UDINT;
	SessionStorage : I_SessionStorage;
	ResponseIdGenerator : I_ResponseIdGenerator;
	HeaderAccessor : I_ChunkedResponseHeaderAccessor;
END_VAR
THIS^.maximumChunkSizeInBytes := MaximumChunkSizeInBytes;
THIS^.maximumPayloadBytesPerChunk := MaximumChunkSizeInBytes - 1;
THIS^.sessionStorage := SessionStorage;
THIS^.responseIdGenerator := ResponseIdGenerator;
This^.headerAccessor := HeaderAccessor;
END_METHOD

METHOD PUBLIC HandleSuccessWithPayload
VAR_INPUT
	OriginalResponse : I_ServerResponse;
	SourceAddress : PVOID;
	SourceSize : UDINT;
END_VAR
VAR
	sessionId : T_MAXSTRING;
	responseId : T_MAXSTRING;
	chunkedResponseData : I_ChunkedResponseData;
END_VAR
IF SourceSize <= maximumPayloadBytesPerChunk THEN
	OriginalResponse.SuccessWithPayload(SourceAddress, SourceSize);
	RETURN;
END_IF

IF NOT headerAccessor.TryGetSessionIdFromResponse(OriginalResponse,sessionId) THEN
	OriginalResponse.Error('MISSING_SESSION_ID','Unable to chunk oversized response without a sessionId');
	RETURN;
END_IF

chunkedResponseData := CreateChunkedResponseData(SourceAddress, SourceSize);
responseId := responseIdGenerator.Generate();

IF NOT sessionStorage.TryStoreSessionDataById(sessionId, responseId, chunkedResponseData) THEN
	OriginalResponse.Error('SERVER_INTERNAL_ERROR','Unable to store oversized response');
	chunkedResponseData.Dispose();
	RETURN;
END_IF

headerAccessor.UpdateResponseWithHasMoreChunks(OriginalResponse, responseId);
chunkedResponseData.SendNextChunk(OriginalResponse, maximumChunkSizeInBytes);
END_METHOD

METHOD PUBLIC TryHandleIncomingRequest : BOOL
VAR_INPUT
	Request : I_Request;
	Response : I_ServerResponse;
END_VAR
VAR
	responseId : T_MAXSTRING;
	sessionId : T_MAXSTRING;
	sessionData : I_SessionData;
	chunkedResponseData : I_ChunkedResponseData;
END_VAR
IF NOT headerAccessor.TryGetResponseIdFromRequest(Request, responseId) THEN
	RETURN;
END_IF

IF NOT headerAccessor.TryGetSessionIdFromRequest(Request, sessionId) THEN
	RETURN;
END_IF

IF NOT sessionStorage.TryRetrieveSessionDataById(sessionId, responseId, sessionData) THEN
	RETURN;
END_IF

IF NOT __QUERYINTERFACE(sessionData, chunkedResponseData) THEN
	RETURN;
END_IF

IF chunkedResponseData.SizeRemaining > maximumPayloadBytesPerChunk THEN
	headerAccessor.UpdateResponseWithHasMoreChunks(Response, responseId);
END_IF

chunkedResponseData.SendNextChunk(Response, maximumChunkSizeInBytes);

IF chunkedResponseData.SendComplete THEN
	sessionStorage.DisposeSessionDataById(sessionId, responseId);
END_IF

TryHandleIncomingRequest := TRUE;
END_METHOD

END_FUNCTION_BLOCK

// ---- mobject-server/_Internal/ChunkedResponses/SessionData/ChunkedResponseData.TcPOU
{attribute 'linkalways'} 
{attribute 'no_explicit_call' := 'This FB is a CLASS and must be accessed using methods or properties'}
{attribute 'enable_dynamic_creation'}
FUNCTION_BLOCK ChunkedResponseData EXTENDS Disposable IMPLEMENTS I_ChunkedResponseData
VAR
	pData : POINTER TO BYTE;
	size : UDINT;
	currentPointerLocation : PVOID;
	remainingLengthToSendInBytes : UDINT;
END_VAR

METHOD FB_exit : BOOL
VAR_INPUT
	bInCopyCode : BOOL; // if TRUE, the exit method is called for exiting an instance that is copied afterwards (online change).
END_VAR
IF bInCopyCode THEN
	RETURN;
END_IF

IF pData <> 0 THEN
	__DELETE(pData);
END_IF
END_METHOD

METHOD FB_init : BOOL
VAR_INPUT
	bInitRetains : BOOL; // if TRUE, the retain variables are initialized (warm start / cold start)
	bInCopyCode : BOOL;  // if TRUE, the instance afterwards gets moved into the copy code (online change)
	Address : PVOID;
	Size : UDINT;
END_VAR
StoreData(Address, Size);
END_METHOD

PROPERTY PUBLIC SendComplete : BOOL
GET
SendComplete := remainingLengthToSendInBytes = 0;
END_GET
END_PROPERTY

METHOD PUBLIC SendNextChunk
VAR_INPUT
	Response : I_ServerResponse;
	Size : UDINT;
END_VAR
VAR
	sendSize : UDINT;
END_VAR
IF SendComplete THEN 
	Response.Error('BAD_REQUEST', 'No further data to send');
	RETURN;
END_IF

sendSize := Size - 1;

IF Size > remainingLengthToSendInBytes THEN 
	sendSize := remainingLengthToSendInBytes;
END_IF

Response.SuccessWithPayload(currentPointerLocation, sendSize);

currentPointerLocation := currentPointerLocation + sendSize;
remainingLengthToSendInBytes := remainingLengthToSendInBytes - sendSize;
END_METHOD

PROPERTY SizeRemaining : UDINT
GET
SizeRemaining := remainingLengthToSendInBytes;
END_GET
END_PROPERTY

METHOD PRIVATE StoreData
VAR_INPUT
	Address : PVOID;
	Size : UDINT;
END_VAR
pData := __NEW(BYTE, Size);
THIS^.size := Size;
memcpy(pData, Address, Size);
currentPointerLocation := pData;
remainingLengthToSendInBytes := Size;
END_METHOD

END_FUNCTION_BLOCK

// ---- mobject-server/_Internal/ChunkedResponses/Middleware/ChunkedResponsesMiddleware.TcPOU
{attribute 'linkalways'} 
{attribute 'no_explicit_call' := 'This FB is a CLASS and must be accessed using methods or properties'}
{attribute 'enable_dynamic_creation'}
FUNCTION_BLOCK ChunkedResponsesMiddleware EXTENDS MiddlewareBase
VAR
	chunkedResponseManager : I_ChunkedResponseManager;
END_VAR

METHOD FB_init : BOOL
VAR_INPUT
	bInitRetains : BOOL; // if TRUE, the retain variables are initialized (warm start / cold start)
	bInCopyCode : BOOL;  // if TRUE, the instance afterwards gets moved into the copy code (online change)
	ChunkedResponseManager : I_ChunkedResponseManager;
END_VAR
THIS^.chunkedResponseManager := ChunkedResponseManager;
END_METHOD

METHOD PUBLIC Handle
VAR_INPUT
	Request : I_Request;
	Response : I_ServerResponse;
END_VAR
VAR
	chunkableServerResponse : ChunkableServerResponse(Response, chunkedResponseManager);
END_VAR
IF chunkedResponseManager.TryHandleIncomingRequest(Request, Response) THEN
	RETURN;
END_IF

Next(Request, chunkableServerResponse);
END_METHOD

END_FUNCTION_BLOCK

// ---- mobject-server/_Internal/ChunkedResponses/ServerResponse/ChunkableServerResponse.TcPOU
{attribute 'linkalways'} 
{attribute 'no_explicit_call' := 'This FB is a CLASS and must be accessed using methods or properties'}
{attribute 'enable_dynamic_creation'}
FUNCTION_BLOCK ChunkableServerResponse IMPLEMENTS I_ServerResponse
VAR
	serverResponse : I_ServerResponse;
	chunkedResponseManager : I_ChunkedResponseManager;
END_VAR

METHOD PUBLIC Accepted
VAR_INPUT
END_VAR
serverResponse.Accepted();
END_METHOD

METHOD PUBLIC Busy
VAR_INPUT
END_VAR
serverResponse.Busy();
END_METHOD

METHOD PUBLIC Error
VAR_INPUT
	ErrorCode : T_MAXSTRING;
	Message : T_MAXSTRING;
END_VAR
serverResponse.Error(ErrorCode, Message);
END_METHOD

METHOD FB_init : BOOL
VAR_INPUT
	bInitRetains : BOOL; // if TRUE, the retain variables are initialized (warm start / cold start)
	bInCopyCode : BOOL;  // if TRUE, the instance afterwards gets moved into the copy code (online change)
	ServerResponse : I_ServerResponse;
	ChunkedResponseManager : I_ChunkedResponseManager;
END_VAR
THIS^.serverResponse := ServerResponse;
This^.chunkedResponseManager := ChunkedResponseManager;
END_METHOD

PROPERTY PUBLIC Header : I_Header
GET
Header := serverResponse.Header;
END_GET
END_PROPERTY

PROPERTY PUBLIC HeadersSent : BOOL
GET
HeadersSent := serverResponse.HeadersSent;
END_GET
END_PROPERTY

METHOD PUBLIC Pending
VAR_INPUT
	ResponseId : REFERENCE TO T_MAXSTRING;
	RetryDelayInMs : UDINT;
END_VAR
serverResponse.Pending(ResponseId, RetryDelayInMs);
END_METHOD

METHOD PUBLIC Success
VAR_INPUT
END_VAR
serverResponse.Success();
END_METHOD

METHOD PUBLIC SuccessWithPayload
VAR_INPUT
	PayloadDataAddress : PVOID;
	PayloadDataSize : UDINT;
END_VAR
chunkedResponseManager.HandleSuccessWithPayload(serverResponse, PayloadDataAddress, PayloadDataSize);
END_METHOD

END_FUNCTION_BLOCK

// ---- mobject-server/_Internal/ServerResponse/ServerResponse.TcPOU
{attribute 'linkalways'} 
{attribute 'no_explicit_call' := 'This FB is a CLASS and must be accessed using methods or properties'}
{attribute 'enable_dynamic_creation'}
FUNCTION_BLOCK ServerResponse IMPLEMENTS I_ServerResponse
VAR
	_header : Header(0);
	_sent : BOOL := FALSE;
	responseData : ResponseData;
	headerAccessor : I_ServerResponseHeaderAccessor;
END_VAR

METHOD PUBLIC Accepted
VAR_INPUT
END_VAR
IF _sent THEN
	RETURN;
END_IF

headerAccessor.UpdateResponseWithAccepted(THIS^);
CompleteResponseWithoutPayload();
END_METHOD

METHOD PUBLIC Busy
VAR_INPUT
END_VAR
IF _sent THEN
	RETURN;
END_IF

headerAccessor.UpdateResponseWithBusy(THIS^);
CompleteResponseWithoutPayload();
END_METHOD

METHOD PRIVATE CompleteResponseWithoutPayload
VAR_INPUT
END_VAR
_sent := TRUE;
_header.ToString(responseData.Header);
memset(ADR(responseData.Payload),0,SIZEOF(responseData.Payload));
END_METHOD

METHOD PRIVATE CompleteResponseWithPayload
VAR_INPUT
	PayloadDataAddress : PVOID;
	PayloadDataSize : UDINT;
END_VAR
_sent := TRUE;
_header.ToString(responseData.Header);
memcpy(ADR(responseData.Payload),PayloadDataAddress,PayloadDataSize);
END_METHOD

METHOD PUBLIC Error
VAR_INPUT
	ErrorCode : T_MAXSTRING;
	Message : T_MAXSTRING;
END_VAR
IF _sent THEN
	RETURN;
END_IF

headerAccessor.UpdateResponseWithError(THIS^, ErrorCode, Message);
CompleteResponseWithoutPayload();
END_METHOD

METHOD FB_init : BOOL
VAR_INPUT
	bInitRetains : BOOL; // if TRUE, the retain variables are initialized (warm start / cold start)
	bInCopyCode : BOOL;  // if TRUE, the instance afterwards gets moved into the copy code (online change)
	HeaderAccessor : I_ServerResponseHeaderAccessor;
END_VAR
THIS^.headerAccessor := HeaderAccessor;
memset(ADR(responseData),0,SIZEOF(responseData));
END_METHOD

PROPERTY PUBLIC Header : I_Header
GET
Header := _header;
END_GET
END_PROPERTY

PROPERTY PUBLIC HeadersSent : BOOL
GET
HeadersSent := _sent;
END_GET
END_PROPERTY

METHOD PUBLIC Pending
VAR_INPUT
	ResponseId : REFERENCE TO T_MAXSTRING;
	RetryDelayInMs : UDINT;
END_VAR
IF _sent THEN
	RETURN;
END_IF

IF (NOT __ISVALIDREF(ResponseId)) OR_ELSE ResponseId = '' THEN
	Error('MISSING_RESPONSE_ID', 'Unable to mark response as pending without ResponseId');
	RETURN;
END_IF

headerAccessor.UpdateResponseWithPending(THIS^, ResponseId, RetryDelayInMs);
CompleteResponseWithoutPayload();
END_METHOD

METHOD PUBLIC Success
VAR_INPUT
END_VAR
VAR
	errorMessage : T_MAXSTRING;
END_VAR
IF _sent THEN
	RETURN;
END_IF

headerAccessor.UpdateResponseWithSuccess(THIS^);
CompleteResponseWithoutPayload();
END_METHOD

METHOD PUBLIC SuccessWithPayload
VAR_INPUT
	PayloadDataAddress : PVOID;
	PayloadDataSize : UDINT;
END_VAR
VAR
	errorMessage : T_MAXSTRING;
	maximumPayloadDataSize : UDINT;
END_VAR
IF _sent THEN
	RETURN;
END_IF

// SIZEOF includes the null terminator, which must stay within the buffer,
// so only SIZEOF - 1 bytes of actual payload data can be transmitted.
maximumPayloadDataSize := SIZEOF(responseData.Payload) - 1;

IF PayloadDataSize > maximumPayloadDataSize THEN
	errorMessage := 'Payload too big to transmit. Maximum : ';
	errorMessage := concat(errorMessage, UDINT_TO_STRING(maximumPayloadDataSize));
	errorMessage := concat(errorMessage, ', Actual Size : ');
	errorMessage := concat(errorMessage, UDINT_TO_STRING(PayloadDataSize));
	Error('PAYLOAD_TOO_BIG', errorMessage);
	RETURN;
END_IF

headerAccessor.UpdateResponseWithSuccess(THIS^);
CompleteResponseWithPayload(PayloadDataAddress, PayloadDataSize);
END_METHOD

METHOD PUBLIC TryGetData : BOOL;
VAR_INPUT
	Destination : REFERENCE TO ResponseData;
END_VAR
IF NOT __ISVALIDREF(Destination) THEN
	RETURN;
END_IF

IF SIZEOF(Destination) <> SIZEOF(responseData) THEN
	RETURN;
END_IF

memcpy(ADR(Destination), ADR(responseData), SIZEOF(Destination));
TryGetData := TRUE;
END_METHOD

END_FUNCTION_BLOCK

// ---- mobject-server/_Internal/AsyncResponse/Manager/AsyncResponseManager.TcPOU
{attribute 'linkalways'} 
{attribute 'no_explicit_call' := 'This FB is a CLASS and must be accessed using methods or properties'}
{attribute 'enable_dynamic_creation'}
FUNCTION_BLOCK AsyncResponseManager IMPLEMENTS I_AsyncResponseManager
VAR
	sessionStorage : I_SessionStorage;
	responseIdGenerator : I_ResponseIdGenerator;
	headerAccessor : I_AsyncResponseHeaderAccessor;
	// how long a handler is given to complete before its pending response is
	// failed.  T#0S disables the deadline.
	pendingResponseMaxAge : TIME;
END_VAR

METHOD PROTECTED CreateAsyncResponseSessionData : I_AsyncResponseSessionData
VAR_INPUT
	RetryDelayInMs : UDINT;
END_VAR
VAR
	pAsyncResponseSessionData : POINTER TO AsyncResponseSessionData;
END_VAR
pAsyncResponseSessionData := __NEW(AsyncResponseSessionData(SuggestedRetryDelayInMs := RetryDelayInMs, MaxAge := pendingResponseMaxAge));
CreateAsyncResponseSessionData := pAsyncResponseSessionData^;
END_METHOD

METHOD PROTECTED CreateAsyncResponseSessionDataProxy : I_AsyncResponseSessionData
VAR_INPUT
	ProxySessionId : T_MAXSTRING;
	ProxyResponseId : T_MAXSTRING;
END_VAR
VAR
	pAsyncResponseSessionDataProxy : POINTER TO AsyncResponseSessionDataProxy;
END_VAR
pAsyncResponseSessionDataProxy := __NEW(AsyncResponseSessionDataProxy(SessionStorage := THIS^.sessionStorage, SessionId := ProxySessionId, ResponseId := ProxyResponseId));
CreateAsyncResponseSessionDataProxy := pAsyncResponseSessionDataProxy^;
END_METHOD

METHOD FB_init : BOOL
VAR_INPUT
	bInitRetains : BOOL; // if TRUE, the retain variables are initialized (warm start / cold start)
	bInCopyCode : BOOL;  // if TRUE, the instance afterwards gets moved into the copy code (online change)
	SessionStorage : I_SessionStorage;
	ResponseIdGenerator : I_ResponseIdGenerator;
	HeaderAccessor : I_AsyncResponseHeaderAccessor;
	PendingResponseMaxAge : TIME;
END_VAR
THIS^.sessionStorage := SessionStorage;
THIS^.responseIdGenerator := ResponseIdGenerator;
THIS^.headerAccessor := HeaderAccessor;
THIS^.pendingResponseMaxAge := PendingResponseMaxAge;
END_METHOD

METHOD TryConvertResponseToAsyncResponseSessionData : BOOL
VAR_INPUT
	Response : I_ServerResponse;
	RetryDelayInMs : UDINT;
	Destination : REFERENCE TO I_AsyncResponseSessionData;
END_VAR
VAR
	sessionId : T_MAXSTRING;
	responseId : T_MAXSTRING;
	newResponseId : T_MAXSTRING;
	asyncResponseSessionData : I_AsyncResponseSessionData;
END_VAR
IF NOT headerAccessor.TryGetSessionIdFromResponse(Response,sessionId) THEN
	Response.Error('MISSING_SESSION_ID','Unable to create a pending response without a sessionId');
	RETURN;
END_IF

asyncResponseSessionData := CreateAsyncResponseSessionData(RetryDelayInMs);
responseId := responseIdGenerator.Generate();

IF NOT sessionStorage.TryStoreSessionDataById(sessionId, responseId, asyncResponseSessionData) THEN
	Response.Error('SERVER_INTERNAL_ERROR','Unable to store pending response');
	asyncResponseSessionData.Dispose();
	RETURN;
END_IF

Response.Pending(responseId, RetryDelayInMs);
Destination := CreateAsyncResponseSessionDataProxy(sessionId, responseId);
TryConvertResponseToAsyncResponseSessionData := true;
END_METHOD

METHOD PUBLIC TryHandleIncomingRequest : BOOL
VAR_INPUT
	Request : I_Request;
	Response : I_ServerResponse;
END_VAR
VAR
	responseId : T_MAXSTRING;
	sessionId : T_MAXSTRING;
	sessionData : I_SessionData;
	asyncResponseData : I_AsyncResponseSessionData;
END_VAR
IF NOT headerAccessor.TryGetResponseIdFromRequest(Request, responseId) THEN
	RETURN;
END_IF

IF NOT headerAccessor.TryGetSessionIdFromRequest(Request, sessionId) THEN
	RETURN;
END_IF

IF NOT sessionStorage.TryRetrieveSessionDataById(sessionId, responseId, sessionData) THEN
	RETURN;
END_IF

IF NOT __QUERYINTERFACE(sessionData, asyncResponseData) THEN
	RETURN;
END_IF

IF asyncResponseData.IsPending THEN

	// The handler was given a deadline and has not completed within it.  Fail the
	// response and discard it rather than telling the client to keep polling - it
	// would otherwise poll forever, and each poll refreshes the session, so the
	// usual session expiry would never reclaim this either.
	IF asyncResponseData.HasExpired THEN
		Response.Error(
			'HANDLER_TIMEOUT',
			'The pending response exceeded its maximum age. The operation may still complete; retry only if it is safe to repeat.'
		);
		sessionStorage.DisposeSessionDataById(sessionId, responseId);
		TryHandleIncomingRequest := TRUE;
		RETURN;
	END_IF

	Response.Pending(responseId, asyncResponseData.SuggestedRetryDelayInMs);
	TryHandleIncomingRequest := TRUE;
	RETURN;
END_IF

IF NOT asyncResponseData.TryUpdateServerResponse(Response) THEN	
	Response.Error('SERVER_INTERNAL_ERROR','Unable to update server response with pending data');
	TryHandleIncomingRequest := TRUE;
	RETURN;
END_IF

sessionStorage.DisposeSessionDataById(sessionId, responseId);
TryHandleIncomingRequest := TRUE;
END_METHOD

END_FUNCTION_BLOCK

// ---- mobject-server/_Internal/AsyncResponse/SessionData/AsyncResponseSessionData.TcPOU
{attribute 'linkalways'} 
{attribute 'no_explicit_call' := 'This FB is a CLASS and must be accessed using methods or properties'}
{attribute 'enable_dynamic_creation'}
FUNCTION_BLOCK AsyncResponseSessionData EXTENDS Disposable IMPLEMENTS I_AsyncResponseSessionData
VAR
	_suggestedRetryDelayInMs : UDINT;
	state : (PENDING, SUCCESS, SUCCESS_WITH_PAYLOAD, ERROR) := PENDING;
	errorCode : T_MAXSTRING;
	errorMessage : T_MAXSTRING;
	pData : POINTER TO BYTE;
	dataSize : UDINT;
	// records the moment this response was created, so the handler can be given
	// a deadline to complete within
	createdTimestamp : SystemTimestamp;
	maxAge : TIME;
END_VAR

METHOD PUBLIC CopyPayloadData
VAR_INPUT
	PayloadDataAddress : PVOID;
	PayloadDataSize : UDINT;
END_VAR
dataSize := PayloadDataSize;
pData := __NEW(BYTE, PayloadDataSize);
memcpy(pData,PayloadDataAddress,PayloadDataSize);
END_METHOD

METHOD PRIVATE DeletePayloadData
VAR_INPUT
END_VAR
IF pData = 0 THEN
	RETURN;
END_IF

__DELETE(pData);
dataSize := 0;
END_METHOD

METHOD PUBLIC Error
VAR_INPUT
	ErrorCode : T_MAXSTRING;
	Message : T_MAXSTRING;
END_VAR
IF state <> PENDING THEN
	RETURN;
END_IF

state := ERROR;
THIS^.errorCode := ErrorCode;
errorMessage := Message;
END_METHOD

METHOD FB_exit : BOOL
VAR_INPUT
	bInCopyCode : BOOL; // if TRUE, the exit method is called for exiting an instance that is copied afterwards (online change).
END_VAR
IF bInCopyCode THEN
	RETURN;
END_IF

DeletePayloadData();
END_METHOD

METHOD FB_init : BOOL
VAR_INPUT
	bInitRetains : BOOL; // if TRUE, the retain variables are initialized (warm start / cold start)
	bInCopyCode : BOOL;  // if TRUE, the instance afterwards gets moved into the copy code (online change)
	SuggestedRetryDelayInMs : UDINT;
	MaxAge : TIME;
END_VAR
_suggestedRetryDelayInMs := SuggestedRetryDelayInMs;
THIS^.maxAge := MaxAge;
END_METHOD

PROPERTY PUBLIC HasExpired : BOOL
GET
// purely a statement about age.  whether that matters is for the caller to
// decide - a response which has already been completed is collectable no
// matter how old it is.
IF maxAge = T#0S THEN
	RETURN;
END_IF

HasExpired := createdTimestamp.IsDurationElapsed(maxAge);
END_GET
END_PROPERTY

PROPERTY PUBLIC IsPending : BOOL
GET
IsPending := state = PENDING;
END_GET
END_PROPERTY

METHOD PUBLIC Success
VAR_INPUT
END_VAR
IF state <> PENDING THEN
	RETURN;
END_IF

state := SUCCESS;
END_METHOD

METHOD PUBLIC SuccessWithPayload
VAR_INPUT
	PayloadDataAddress : PVOID;
	PayloadDataSize : UDINT;
END_VAR
IF state <> PENDING THEN
	RETURN;
END_IF

state := SUCCESS_WITH_PAYLOAD;
CopyPayloadData(PayloadDataAddress, PayloadDataSize);
END_METHOD

PROPERTY PUBLIC SuggestedRetryDelayInMs : UDINT
GET
SuggestedRetryDelayInMs := _suggestedRetryDelayInMs;
END_GET
SET // PUBLIC
_suggestedRetryDelayInMs := SuggestedRetryDelayInMs;
END_SET
END_PROPERTY

METHOD PUBLIC TryUpdateServerResponse : BOOL
VAR_INPUT
	Response : I_ServerResponse;
END_VAR
IF State = SUCCESS_WITH_PAYLOAD THEN
	Response.SuccessWithPayload(pData,dataSize);
	TryUpdateServerResponse := TRUE;
	RETURN;
END_IF

IF State = SUCCESS THEN
	Response.Success();
	TryUpdateServerResponse := TRUE;
	RETURN;
END_IF

IF state = ERROR THEN
	Response.Error(errorCode, errorMessage);
	TryUpdateServerResponse := TRUE;
	RETURN;
END_IF
END_METHOD

END_FUNCTION_BLOCK

// ---- mobject-server/_Internal/AsyncResponse/Proxy/AsyncResponseSessionDataProxy.TcPOU
{attribute 'linkalways'} 
{attribute 'no_explicit_call' := 'This FB is a CLASS and must be accessed using methods or properties'}
{attribute 'enable_dynamic_creation'}
FUNCTION_BLOCK AsyncResponseSessionDataProxy EXTENDS Disposable IMPLEMENTS I_AsyncResponseSessionData
VAR
	sessionStorage : I_SessionStorage;
	sessionId : T_MAXSTRING;
	responseId : T_MAXSTRING;
END_VAR

METHOD PUBLIC Error
VAR_INPUT
	ErrorCode : T_MAXSTRING;
	Message : T_MAXSTRING;
END_VAR
VAR
	asyncReponseSessionData : I_AsyncResponseSessionData;
END_VAR
IF NOT TryGetAsyncResponseSessionData(asyncReponseSessionData) THEN
	RETURN;
END_IF

asyncReponseSessionData.Error(ErrorCode, Message);
END_METHOD

METHOD FB_init : BOOL
VAR_INPUT
	bInitRetains : BOOL; // if TRUE, the retain variables are initialized (warm start / cold start)
	bInCopyCode : BOOL;  // if TRUE, the instance afterwards gets moved into the copy code (online change)
	SessionStorage : I_SessionStorage;
	SessionId : T_MAXSTRING;
	ResponseId : T_MAXSTRING;
END_VAR
THIS^.sessionStorage := SessionStorage;
THIS^.sessionId := SessionId;
THIS^.responseId := ResponseId;
END_METHOD

PROPERTY PUBLIC HasExpired : BOOL
GET
VAR
	asyncReponseSessionData : I_AsyncResponseSessionData;
END_VAR
IF NOT TryGetAsyncResponseSessionData(asyncReponseSessionData) THEN
	RETURN;
END_IF

HasExpired := asyncReponseSessionData.HasExpired;
END_GET
END_PROPERTY

PROPERTY PUBLIC IsPending : BOOL
GET
VAR
	asyncReponseSessionData : I_AsyncResponseSessionData;
END_VAR
IF NOT TryGetAsyncResponseSessionData(asyncReponseSessionData) THEN
	RETURN;
END_IF

IsPending := asyncReponseSessionData.IsPending;
END_GET
END_PROPERTY

METHOD PUBLIC Success
VAR_INPUT
END_VAR
VAR
	asyncReponseSessionData : I_AsyncResponseSessionData;
END_VAR
IF NOT TryGetAsyncResponseSessionData(asyncReponseSessionData) THEN
	RETURN;
END_IF

asyncReponseSessionData.Success();
END_METHOD

METHOD PUBLIC SuccessWithPayload
VAR_INPUT
	PayloadDataAddress : PVOID;
	PayloadDataSize : UDINT;
END_VAR
VAR
	asyncReponseSessionData : I_AsyncResponseSessionData;
END_VAR
IF NOT TryGetAsyncResponseSessionData(asyncReponseSessionData) THEN
	RETURN;
END_IF

asyncReponseSessionData.SuccessWithPayload(PayloadDataAddress, PayloadDataSize);
END_METHOD

PROPERTY PUBLIC SuggestedRetryDelayInMs : UDINT
GET
VAR
	asyncReponseSessionData : I_AsyncResponseSessionData;
END_VAR
IF NOT TryGetAsyncResponseSessionData(asyncReponseSessionData) THEN
	RETURN;
END_IF

SuggestedRetryDelayInMs := asyncReponseSessionData.SuggestedRetryDelayInMs;
END_GET
SET // PUBLIC
VAR
	asyncReponseSessionData : I_AsyncResponseSessionData;
END_VAR
IF NOT TryGetAsyncResponseSessionData(asyncReponseSessionData) THEN
	RETURN;
END_IF

asyncReponseSessionData.SuggestedRetryDelayInMs := SuggestedRetryDelayInMs;
END_SET
END_PROPERTY

METHOD PROTECTED TryGetAsyncResponseSessionData : BOOL;
VAR_INPUT
	Destination : REFERENCE TO I_AsyncResponseSessionData;
END_VAR
VAR
	sessionData : I_SessionData;
	asyncSessionData : I_AsyncResponseSessionData;
END_VAR
IF NOT sessionStorage.TryRetrieveSessionDataById(sessionId, responseId, sessionData) THEN
	RETURN;
END_IF

IF NOT __QUERYINTERFACE(sessionData, asyncSessionData) THEN
	RETURN;
END_IF

Destination := asyncSessionData;
TryGetAsyncResponseSessionData := TRUE;
END_METHOD

METHOD PUBLIC TryUpdateServerResponse : BOOL
VAR_INPUT
	Response : I_ServerResponse;
END_VAR
VAR
	asyncReponseSessionData : I_AsyncResponseSessionData;
END_VAR
IF NOT TryGetAsyncResponseSessionData(asyncReponseSessionData) THEN
	RETURN;
END_IF

TryUpdateServerResponse := asyncReponseSessionData.TryUpdateServerResponse(Response);
END_METHOD

END_FUNCTION_BLOCK

// ---- mobject-server/_Internal/AsyncResponse/Middleware/AsyncResponseMiddleware.TcPOU
FUNCTION_BLOCK AsyncResponseMiddleware EXTENDS MiddlewareBase
VAR
	asyncResponseManager : I_AsyncResponseManager;
END_VAR

METHOD FB_init : BOOL
VAR_INPUT
	bInitRetains : BOOL; // if TRUE, the retain variables are initialized (warm start / cold start)
	bInCopyCode : BOOL;  // if TRUE, the instance afterwards gets moved into the copy code (online change)
	AsyncResponseManager : I_AsyncResponseManager;
END_VAR
This^.asyncResponseManager := AsyncResponseManager;
END_METHOD

METHOD PUBLIC Handle
VAR_INPUT
	Request : I_Request;
	Response : I_ServerResponse;
END_VAR
IF asyncResponseManager.TryHandleIncomingRequest(Request, Response) THEN
	RETURN;
END_IF

Next(Request, Response);
END_METHOD

END_FUNCTION_BLOCK

// ---- mobject-server/_Internal/Followup/Middleware/ResponseIdGuardMiddleware.TcPOU
{attribute 'linkalways'} 
{attribute 'no_explicit_call' := 'This FB is a CLASS and must be accessed using methods or properties'}
{attribute 'enable_dynamic_creation'}
FUNCTION_BLOCK ResponseIdGuardMiddleware EXTENDS MiddlewareBase
VAR
	headerAccessor : I_SessionHeaderAccessor;
END_VAR

METHOD FB_init : BOOL
VAR_INPUT
	bInitRetains : BOOL; // if TRUE, the retain variables are initialized (warm start / cold start)
	bInCopyCode : BOOL;  // if TRUE, the instance afterwards gets moved into the copy code (online change)
	HeaderAccessor : I_SessionHeaderAccessor;
END_VAR
THIS^.headerAccessor := HeaderAccessor;
END_METHOD

